LIN {X 0,Y 290.409,Z 885.238,A -85,B 0,C 180,E1 14491.775,E2 14491.775} C_VEL
LIN {X 0,Y 290.448,Z 885.193,A -85,B 0,C 180,E1 14487.632,E2 14487.632} C_VEL
LIN {X 0,Y 290.881,Z 883.624,A -85,B 0,C 180,E1 14483.487,E2 14483.487} C_VEL
LIN {X 0,Y 291.889,Z 880.575,A -85,B 0,C 180,E1 14479.341,E2 14479.341} C_VEL
LIN {X 0,Y 293.714,Z 875.67,A -85,B 0,C 180,E1 14475.007,E2 14475.007} C_VEL
LIN {X 0,Y 296.27,Z 869.554,A -85,B 0,C 180,E1 14471.097,E2 14471.097} C_VEL
LIN {X 0,Y 299.729,Z 861.682,A -85,B 0,C 180,E1 14467.236,E2 14467.236} C_VEL
LIN {X 0,Y 304.292,Z 851.484,A -85,B 0,C 180,E1 14463.349,E2 14463.349} C_VEL
LIN {X 0,Y 309.291,Z 840.18,A -85,B 0,C 180,E1 14459.931,E2 14459.931} C_VEL
LIN {X 0,Y 314.618,Z 827.702,A -85,B 0,C 180,E1 14456.868,E2 14456.868} C_VEL
LIN {X 0,Y 320.27,Z 813.754,A -85,B 0,C 180,E1 14454.065,E2 14454.065} C_VEL
LIN {X 0,Y 325.878,Z 798.802,A -85,B 0,C 180,E1 14451.592,E2 14451.592} C_VEL
LIN {X 0,Y 326.277,Z 797.642,A -85,B 0,C 180,E1 14451.422,E2 14451.422} C_VEL
LIN {X 0,Y 327.524,Z 792.143,A -85,B 0,C 180,E1 14450.493,E2 14450.493} C_VEL
LIN {X 0,Y 328.002,Z 778.328,A -85,B 0,C 180,E1 14447.929,E2 14447.929} C_VEL
LIN {X 0,Y 329.187,Z 772.235,A -85,B 0,C 180,E1 14447.122,E2 14447.122} C_VEL
LIN {X 0,Y 334.318,Z 754.064,A -85,B 0,C 180,E1 14445.351,E2 14445.351} C_VEL
LIN {X 0,Y 338.615,Z 735.624,A -85,B 0,C 180,E1 14443.911,E2 14443.911} C_VEL
LIN {X 0,Y 342.229,Z 716.359,A -85,B 0,C 180,E1 14442.716,E2 14442.716} C_VEL
LIN {X 0,Y 345.103,Z 695.919,A -85,B 0,C 180,E1 14441.743,E2 14441.743} C_VEL
LIN {X 0,Y 346.998,Z 675.756,A -85,B 0,C 180,E1 14441.046,E2 14441.046} C_VEL
LIN {X 0,Y 349.676,Z 625.674,A -85,B 0,C 180,E1 14439.978,E2 14439.978} C_VEL
LIN {X 0,Y 357.062,Z 493.743,A -85,B 0,C 180,E1 14437.345,E2 14437.345} C_VEL
LIN {X 0,Y 348.869,Z 480.651,A -85,B 0,C 180,E1 14434.824,E2 14434.824} C_VEL
LIN {X 0,Y 340.95,Z 468.944,A -85,B 0,C 180,E1 14432.109,E2 14432.109} C_VEL
LIN {X 0,Y 333.261,Z 458.594,A -85,B 0,C 180,E1 14429.13,E2 14429.13} C_VEL
LIN {X 0,Y 329.157,Z 453.339,A -85,B 0,C 180,E1 14427.352,E2 14427.352} C_VEL
LIN {X 0,Y 325.768,Z 449.026,A -85,B 0,C 180,E1 14425.741,E2 14425.741} C_VEL
LIN {X 0,Y 321.751,Z 444.067,A -85,B 0,C 180,E1 14423.633,E2 14423.633} C_VEL
LIN {X 0,Y 317.156,Z 438.642,A -85,B 0,C 180,E1 14420.87,E2 14420.87} C_VEL
LIN {X 0,Y 313.204,Z 434.22,A -85,B 0,C 180,E1 14418.039,E2 14418.039} C_VEL
LIN {X 0,Y 311.897,Z 432.781,A -85,B 0,C 180,E1 14416.961,E2 14416.961} C_VEL
LIN {X 0,Y 306.235,Z 426.851,A -85,B 0,C 180,E1 14410.536,E2 14410.536} C_VEL
LIN {X 0,Y 304.093,Z 425.512,A -85,B 0,C 180,E1 14405.012,E2 14405.012} C_VEL
LIN {X 0,Y 304.604,Z 426.367,A -85,B 0,C 180,E1 14399.248,E2 14399.248} C_VEL
LIN {X 0,Y 308.994,Z 432.434,A -85,B 0,C 180,E1 14392.096,E2 14392.096} C_VEL
LIN {X 0,Y 312.085,Z 436.892,A -85,B 0,C 180,E1 14389.105,E2 14389.105} C_VEL
LIN {X 0,Y 313.416,Z 438.523,A -85,B 0,C 180,E1 14388.033,E2 14388.033} C_VEL
LIN {X 0,Y 317.449,Z 443.877,A -85,B 0,C 180,E1 14385.173,E2 14385.173} C_VEL
LIN {X 0,Y 322.042,Z 450.238,A -85,B 0,C 180,E1 14382.427,E2 14382.427} C_VEL
LIN {X 0,Y 325.886,Z 455.636,A -85,B 0,C 180,E1 14380.416,E2 14380.416} C_VEL
LIN {X 0,Y 329.975,Z 461.384,A -85,B 0,C 180,E1 14378.492,E2 14378.492} C_VEL
LIN {X 0,Y 337.184,Z 472.131,A -85,B 0,C 180,E1 14375.472,E2 14375.472} C_VEL
LIN {X 0,Y 345.291,Z 485.16,A -85,B 0,C 180,E1 14372.493,E2 14372.493} C_VEL
LIN {X 0,Y 353.679,Z 499.744,A -85,B 0,C 180,E1 14369.741,E2 14369.741} C_VEL
LIN {X 0,Y 358.79,Z 509.616,A -85,B 0,C 180,E1 14368.177,E2 14368.177} C_VEL
LIN {X 0,Y 345.156,Z 726.934,A -85,B 0,C 180,E1 14363.563,E2 14363.563} C_VEL
LIN {X 0,Y 342.592,Z 750.271,A -85,B 0,C 180,E1 14362.89,E2 14362.89} C_VEL
LIN {X 0,Y 339.061,Z 771.428,A -85,B 0,C 180,E1 14362.078,E2 14362.078} C_VEL
LIN {X 0,Y 334.52,Z 792.579,A -85,B 0,C 180,E1 14360.992,E2 14360.992} C_VEL
LIN {X 0,Y 329.38,Z 812.962,A -85,B 0,C 180,E1 14359.629,E2 14359.629} C_VEL
LIN {X 0,Y 323.471,Z 833.709,A -85,B 0,C 180,E1 14357.875,E2 14357.875} C_VEL
LIN {X 0,Y 317.514,Z 852.768,A -85,B 0,C 180,E1 14355.883,E2 14355.883} C_VEL
LIN {X 0,Y 311.126,Z 871.664,A -85,B 0,C 180,E1 14353.446,E2 14353.446} C_VEL
LIN {X 0,Y 305.032,Z 889.034,A -85,B 0,C 180,E1 14350.711,E2 14350.711} C_VEL
LIN {X 0,Y 298.988,Z 905.992,A -85,B 0,C 180,E1 14347.487,E2 14347.487} C_VEL
LIN {X 0,Y 293.913,Z 920.626,A -85,B 0,C 180,E1 14344.143,E2 14344.143} C_VEL
LIN {X 0,Y 289.56,Z 933.897,A -85,B 0,C 180,E1 14340.501,E2 14340.501} C_VEL
LIN {X 0,Y 286.009,Z 946,A -85,B 0,C 180,E1 14336.499,E2 14336.499} C_VEL
LIN {X 0,Y 283.419,Z 956.775,A -85,B 0,C 180,E1 14332.176,E2 14332.176} C_VEL
LIN {X 0,Y 281.949,Z 965.312,A -85,B 0,C 180,E1 14327.969,E2 14327.969} C_VEL
LIN {X 0,Y 281.351,Z 971.642,A -85,B 0,C 180,E1 14323.984,E2 14323.984} C_VEL
LIN {X 0,Y 281.318,Z 976.689,A -85,B 0,C 180,E1 14319.822,E2 14319.822} C_VEL
LIN {X 0,Y 281.574,Z 979.725,A -85,B 0,C 180,E1 14316.115,E2 14316.115} C_VEL
LIN {X 0,Y 281.797,Z 981.427,A -85,B 0,C 180,E1 14312.441,E2 14312.441} C_VEL
LIN {X 0,Y 281.86,Z 981.636,A -85,B 0,C 180,E1 14308.985,E2 14308.985} C_VEL
LIN {X 0,Y 281.703,Z 980.723,A -85,B 0,C 180,E1 14305.727,E2 14305.727} C_VEL
LIN {X 0,Y 281.41,Z 978.219,A -85,B 0,C 180,E1 14301.831,E2 14301.831} C_VEL
LIN {X 0,Y 281.285,Z 974.359,A -85,B 0,C 180,E1 14298.104,E2 14298.104} C_VEL
LIN {X 0,Y 281.594,Z 968.491,A -85,B 0,C 180,E1 14293.924,E2 14293.924} C_VEL
LIN {X 0,Y 282.637,Z 960.839,A -85,B 0,C 180,E1 14289.718,E2 14289.718} C_VEL
LIN {X 0,Y 284.644,Z 951.268,A -85,B 0,C 180,E1 14285.516,E2 14285.516} C_VEL
LIN {X 0,Y 287.76,Z 939.735,A -85,B 0,C 180,E1 14281.351,E2 14281.351} C_VEL
LIN {X 0,Y 291.612,Z 927.517,A -85,B 0,C 180,E1 14277.669,E2 14277.669} C_VEL
LIN {X 0,Y 296.576,Z 912.818,A -85,B 0,C 180,E1 14274.009,E2 14274.009} C_VEL
LIN {X 0,Y 302.138,Z 897.046,A -85,B 0,C 180,E1 14270.747,E2 14270.747} C_VEL
LIN {X 0,Y 308.386,Z 879.4,A -85,B 0,C 180,E1 14267.726,E2 14267.726} C_VEL
LIN {X 0,Y 314.378,Z 862.063,A -85,B 0,C 180,E1 14265.267,E2 14265.267} C_VEL
LIN {X 0,Y 320.426,Z 843.454,A -85,B 0,C 180,E1 14263.106,E2 14263.106} C_VEL
LIN {X 0,Y 326.091,Z 824.547,A -85,B 0,C 180,E1 14261.312,E2 14261.312} C_VEL
LIN {X 0,Y 331.598,Z 804.213,A -85,B 0,C 180,E1 14259.753,E2 14259.753} C_VEL
LIN {X 0,Y 336.584,Z 783.168,A -85,B 0,C 180,E1 14258.495,E2 14258.495} C_VEL
LIN {X 0,Y 340.77,Z 761.554,A -85,B 0,C 180,E1 14257.53,E2 14257.53} C_VEL
LIN {X 0,Y 343.932,Z 738.988,A -85,B 0,C 180,E1 14256.768,E2 14256.768} C_VEL
LIN {X 0,Y 346.033,Z 712.945,A -85,B 0,C 180,E1 14256.132,E2 14256.132} C_VEL
LIN {X 0,Y 358.699,Z 509.365,A -85,B 0,C 180,E1 14251.827,E2 14251.827} C_VEL
LIN {X 0,Y 349.918,Z 493.137,A -85,B 0,C 180,E1 14249.109,E2 14249.109} C_VEL
LIN {X 0,Y 341.866,Z 479.602,A -85,B 0,C 180,E1 14246.348,E2 14246.348} C_VEL
LIN {X 0,Y 335.259,Z 469.393,A -85,B 0,C 180,E1 14243.835,E2 14243.835} C_VEL
LIN {X 0,Y 327.618,Z 457.902,A -85,B 0,C 180,E1 14240.499,E2 14240.499} C_VEL
LIN {X 0,Y 320.59,Z 448.147,A -85,B 0,C 180,E1 14236.86,E2 14236.86} C_VEL
LIN {X 0,Y 316.137,Z 442.173,A -85,B 0,C 180,E1 14234.095,E2 14234.095} C_VEL
LIN {X 0,Y 312.318,Z 437.185,A -85,B 0,C 180,E1 14231.261,E2 14231.261} C_VEL
LIN {X 0,Y 309.021,Z 432.656,A -85,B 0,C 180,E1 14228.184,E2 14228.184} C_VEL
LIN {X 0,Y 308.029,Z 431.411,A -85,B 0,C 180,E1 14227.085,E2 14227.085} C_VEL
LIN {X 0,Y 304.423,Z 426.254,A -85,B 0,C 180,E1 14220.941,E2 14220.941} C_VEL
LIN {X 0,Y 303.838,Z 425.332,A -85,B 0,C 180,E1 14214.902,E2 14214.902} C_VEL
LIN {X 0,Y 305.725,Z 426.487,A -85,B 0,C 180,E1 14209.828,E2 14209.828} C_VEL
LIN {X 0,Y 307.208,Z 427.964,A -85,B 0,C 180,E1 14207.595,E2 14207.595} C_VEL
LIN {X 0,Y 312.808,Z 433.677,A -85,B 0,C 180,E1 14202.034,E2 14202.034} C_VEL
LIN {X 0,Y 316.844,Z 438.399,A -85,B 0,C 180,E1 14199.109,E2 14199.109} C_VEL
LIN {X 0,Y 318.218,Z 439.909,A -85,B 0,C 180,E1 14198.237,E2 14198.237} C_VEL
LIN {X 0,Y 322.234,Z 444.497,A -85,B 0,C 180,E1 14195.918,E2 14195.918} C_VEL
LIN {X 0,Y 327.796,Z 451.607,A -85,B 0,C 180,E1 14193.115,E2 14193.115} C_VEL
LIN {X 0,Y 332.097,Z 457.141,A -85,B 0,C 180,E1 14191.202,E2 14191.202} C_VEL
LIN {X 0,Y 338.239,Z 465.249,A -85,B 0,C 180,E1 14188.748,E2 14188.748} C_VEL
LIN {X 0,Y 346.862,Z 477.634,A -85,B 0,C 180,E1 14185.698,E2 14185.698} C_VEL
LIN {X 0,Y 355.474,Z 491.21,A -85,B 0,C 180,E1 14182.992,E2 14182.992} C_VEL
LIN {X 0,Y 357.054,Z 494.161,A -85,B 0,C 180,E1 14182.515,E2 14182.515} C_VEL
LIN {X 0,Y 347.059,Z 672.789,A -85,B 0,C 180,E1 14178.93,E2 14178.93} C_VEL
LIN {X 0,Y 345.224,Z 693.984,A -85,B 0,C 180,E1 14178.232,E2 14178.232} C_VEL
LIN {X 0,Y 342.488,Z 714.257,A -85,B 0,C 180,E1 14177.297,E2 14177.297} C_VEL
LIN {X 0,Y 339.005,Z 733.494,A -85,B 0,C 180,E1 14176.136,E2 14176.136} C_VEL
LIN {X 0,Y 334.567,Z 752.673,A -85,B 0,C 180,E1 14174.661,E2 14174.661} C_VEL
LIN {X 0,Y 329.766,Z 769.978,A -85,B 0,C 180,E1 14173.01,E2 14173.01} C_VEL
LIN {X 0,Y 324.127,Z 787.653,A -85,B 0,C 180,E1 14170.941,E2 14170.941} C_VEL
LIN {X 0,Y 318.438,Z 803.532,A -85,B 0,C 180,E1 14168.665,E2 14168.665} C_VEL
LIN {X 0,Y 312.517,Z 818.483,A -85,B 0,C 180,E1 14166.059,E2 14166.059} C_VEL
LIN {X 0,Y 306.776,Z 831.838,A -85,B 0,C 180,E1 14163.195,E2 14163.195} C_VEL
LIN {X 0,Y 301.346,Z 843.808,A -85,B 0,C 180,E1 14160.063,E2 14160.063} C_VEL
LIN {X 0,Y 296.149,Z 854.942,A -85,B 0,C 180,E1 14156.462,E2 14156.462} C_VEL
LIN {X 0,Y 291.874,Z 864.064,A -85,B 0,C 180,E1 14152.771,E2 14152.771} C_VEL
LIN {X 0,Y 288.37,Z 871.774,A -85,B 0,C 180,E1 14148.809,E2 14148.809} C_VEL
LIN {X 0,Y 285.67,Z 877.943,A -85,B 0,C 180,E1 14144.594,E2 14144.594} C_VEL
LIN {X 0,Y 283.939,Z 882.349,A -85,B 0,C 180,E1 14140.344,E2 14140.344} C_VEL
LIN {X 0,Y 282.94,Z 885.19,A -85,B 0,C 180,E1 14136.084,E2 14136.084} C_VEL
LIN {X 0,Y 282.523,Z 886.567,A -85,B 0,C 180,E1 14131.824,E2 14131.824} C_VEL
LIN {X 0,Y 282.563,Z 886.521,A -85,B 0,C 180,E1 14127.566,E2 14127.566} C_VEL
LIN {X 0,Y 283.03,Z 884.955,A -85,B 0,C 180,E1 14123.305,E2 14123.305} C_VEL
LIN {X 0,Y 284.108,Z 881.909,A -85,B 0,C 180,E1 14119.045,E2 14119.045} C_VEL
LIN {X 0,Y 286.058,Z 877.01,A -85,B 0,C 180,E1 14114.596,E2 14114.596} C_VEL
LIN {X 0,Y 288.767,Z 870.9,A -85,B 0,C 180,E1 14110.587,E2 14110.587} C_VEL
LIN {X 0,Y 292.425,Z 863.031,A -85,B 0,C 180,E1 14106.634,E2 14106.634} C_VEL
LIN {X 0,Y 297.085,Z 853.112,A -85,B 0,C 180,E1 14102.762,E2 14102.762} C_VEL
LIN {X 0,Y 302.17,Z 842.154,A -85,B 0,C 180,E1 14099.353,E2 14099.353} C_VEL
LIN {X 0,Y 307.678,Z 829.872,A -85,B 0,C 180,E1 14096.244,E2 14096.244} C_VEL
LIN {X 0,Y 313.527,Z 816.113,A -85,B 0,C 180,E1 14093.394,E2 14093.394} C_VEL
LIN {X 0,Y 319.335,Z 801.393,A -85,B 0,C 180,E1 14090.887,E2 14090.887} C_VEL
LIN {X 0,Y 325.122,Z 785.032,A -85,B 0,C 180,E1 14088.613,E2 14088.613} C_VEL
LIN {X 0,Y 329.187,Z 772.235,A -85,B 0,C 180,E1 14087.122,E2 14087.122} C_VEL
LIN {X 0,Y 330.457,Z 765.992,A -85,B 0,C 180,E1 14086.346,E2 14086.346} C_VEL
LIN {X 0,Y 330.75,Z 750.626,A -85,B 0,C 180,E1 14084.094,E2 14084.094} C_VEL
LIN {X 0,Y 331.712,Z 743.976,A -85,B 0,C 180,E1 14083.429,E2 14083.429} C_VEL
LIN {X 0,Y 335.725,Z 725.177,A -85,B 0,C 180,E1 14082.14,E2 14082.14} C_VEL
LIN {X 0,Y 338.968,Z 705.436,A -85,B 0,C 180,E1 14081.084,E2 14081.084} C_VEL
LIN {X 0,Y 341.414,Z 684.411,A -85,B 0,C 180,E1 14080.253,E2 14080.253} C_VEL
LIN {X 0,Y 342.879,Z 662.381,A -85,B 0,C 180,E1 14079.658,E2 14079.658} C_VEL
LIN {X 0,Y 352.377,Z 497.735,A -85,B 0,C 180,E1 14076.345,E2 14076.345} C_VEL
LIN {X 0,Y 343.887,Z 484.113,A -85,B 0,C 180,E1 14073.584,E2 14073.584} C_VEL
LIN {X 0,Y 335.378,Z 471.633,A -85,B 0,C 180,E1 14070.453,E2 14070.453} C_VEL
LIN {X 0,Y 327.784,Z 461.467,A -85,B 0,C 180,E1 14067.23,E2 14067.23} C_VEL
LIN {X 0,Y 323.657,Z 456.225,A -85,B 0,C 180,E1 14065.234,E2 14065.234} C_VEL
LIN {X 0,Y 319.892,Z 451.487,A -85,B 0,C 180,E1 14063.193,E2 14063.193} C_VEL
LIN {X 0,Y 315.547,Z 446.233,A -85,B 0,C 180,E1 14060.496,E2 14060.496} C_VEL
LIN {X 0,Y 311.599,Z 441.616,A -85,B 0,C 180,E1 14057.556,E2 14057.556} C_VEL
LIN {X 0,Y 309.905,Z 440.067,A -85,B 0,C 180,E1 14056.109,E2 14056.109} C_VEL
LIN {X 0,Y 305.169,Z 434.743,A -85,B 0,C 180,E1 14050.382,E2 14050.382} C_VEL
LIN {X 0,Y 303.105,Z 433.451,A -85,B 0,C 180,E1 14044.921,E2 14044.921} C_VEL
LIN {X 0,Y 303.611,Z 434.332,A -85,B 0,C 180,E1 14039.246,E2 14039.246} C_VEL
LIN {X 0,Y 307.728,Z 440.294,A -85,B 0,C 180,E1 14032.345,E2 14032.345} C_VEL
LIN {X 0,Y 310.977,Z 444.898,A -85,B 0,C 180,E1 14029.159,E2 14029.159} C_VEL
LIN {X 0,Y 315.697,Z 451.327,A -85,B 0,C 180,E1 14025.605,E2 14025.605} C_VEL
LIN {X 0,Y 320.403,Z 458.009,A -85,B 0,C 180,E1 14022.709,E2 14022.709} C_VEL
LIN {X 0,Y 325.963,Z 465.865,A -85,B 0,C 180,E1 14019.814,E2 14019.814} C_VEL
LIN {X 0,Y 333.477,Z 477.362,A -85,B 0,C 180,E1 14016.452,E2 14016.452} C_VEL
LIN {X 0,Y 339.968,Z 487.805,A -85,B 0,C 180,E1 14013.917,E2 14013.917} C_VEL
LIN {X 0,Y 347.35,Z 500.6,A -85,B 0,C 180,E1 14011.315,E2 14011.315} C_VEL
LIN {X 0,Y 353.993,Z 513.293,A -85,B 0,C 180,E1 14009.161,E2 14009.161} C_VEL
LIN {X 0,Y 340.097,Z 726.961,A -85,B 0,C 180,E1 14004.602,E2 14004.602} C_VEL
LIN {X 0,Y 337.422,Z 750.06,A -85,B 0,C 180,E1 14003.925,E2 14003.925} C_VEL
LIN {X 0,Y 333.61,Z 771.835,A -85,B 0,C 180,E1 14003.073,E2 14003.073} C_VEL
LIN {X 0,Y 328.817,Z 793.371,A -85,B 0,C 180,E1 14001.952,E2 14001.952} C_VEL
LIN {X 0,Y 323.524,Z 813.342,A -85,B 0,C 180,E1 14000.585,E2 14000.585} C_VEL
LIN {X 0,Y 317.443,Z 833.743,A -85,B 0,C 180,E1 13998.826,E2 13998.826} C_VEL
LIN {X 0,Y 311.264,Z 852.623,A -85,B 0,C 180,E1 13996.813,E2 13996.813} C_VEL
LIN {X 0,Y 304.638,Z 871.415,A -85,B 0,C 180,E1 13994.349,E2 13994.349} C_VEL
LIN {X 0,Y 298.296,Z 888.614,A -85,B 0,C 180,E1 13991.577,E2 13991.577} C_VEL
LIN {X 0,Y 292.146,Z 904.974,A -85,B 0,C 180,E1 13988.396,E2 13988.396} C_VEL
LIN {X 0,Y 286.666,Z 919.933,A -85,B 0,C 180,E1 13984.888,E2 13984.888} C_VEL
LIN {X 0,Y 282.089,Z 933.143,A -85,B 0,C 180,E1 13981.162,E2 13981.162} C_VEL
LIN {X 0,Y 278.396,Z 944.932,A -85,B 0,C 180,E1 13977.135,E2 13977.135} C_VEL
LIN {X 0,Y 275.596,Z 955.82,A -85,B 0,C 180,E1 13972.615,E2 13972.615} C_VEL
LIN {X 0,Y 274.039,Z 964.27,A -85,B 0,C 180,E1 13968.286,E2 13968.286} C_VEL
LIN {X 0,Y 273.401,Z 970.56,A -85,B 0,C 180,E1 13964.183,E2 13964.183} C_VEL
LIN {X 0,Y 273.386,Z 975.525,A -85,B 0,C 180,E1 13959.898,E2 13959.898} C_VEL
LIN {X 0,Y 273.641,Z 978.381,A -85,B 0,C 180,E1 13956.293,E2 13956.293} C_VEL
LIN {X 0,Y 273.901,Z 980.097,A -85,B 0,C 180,E1 13952.511,E2 13952.511} C_VEL
LIN {X 0,Y 273.971,Z 980.307,A -85,B 0,C 180,E1 13948.955,E2 13948.955} C_VEL
LIN {X 0,Y 273.789,Z 979.36,A -85,B 0,C 180,E1 13945.537,E2 13945.537} C_VEL
LIN {X 0,Y 273.466,Z 976.864,A -85,B 0,C 180,E1 13941.592,E2 13941.592} C_VEL
LIN {X 0,Y 273.34,Z 972.987,A -85,B 0,C 180,E1 13937.753,E2 13937.753} C_VEL
LIN {X 0,Y 273.736,Z 966.743,A -85,B 0,C 180,E1 13933.231,E2 13933.231} C_VEL
LIN {X 0,Y 274.932,Z 959.016,A -85,B 0,C 180,E1 13928.901,E2 13928.901} C_VEL
LIN {X 0,Y 277.167,Z 949.314,A -85,B 0,C 180,E1 13924.582,E2 13924.582} C_VEL
LIN {X 0,Y 280.579,Z 937.642,A -85,B 0,C 180,E1 13920.312,E2 13920.312} C_VEL
LIN {X 0,Y 285.012,Z 924.508,A -85,B 0,C 180,E1 13916.343,E2 13916.343} C_VEL
LIN {X 0,Y 290.333,Z 909.936,A -85,B 0,C 180,E1 13912.696,E2 13912.696} C_VEL
LIN {X 0,Y 296.32,Z 893.776,A -85,B 0,C 180,E1 13909.371,E2 13909.371} C_VEL
LIN {X 0,Y 302.646,Z 876.69,A -85,B 0,C 180,E1 13906.469,E2 13906.469} C_VEL
LIN {X 0,Y 309.294,Z 858.127,A -85,B 0,C 180,E1 13903.878,E2 13903.878} C_VEL
LIN {X 0,Y 315.572,Z 839.508,A -85,B 0,C 180,E1 13901.749,E2 13901.749} C_VEL
LIN {X 0,Y 321.813,Z 819.166,A -85,B 0,C 180,E1 13899.885,E2 13899.885} C_VEL
LIN {X 0,Y 327.168,Z 799.467,A -85,B 0,C 180,E1 13898.45,E2 13898.45} C_VEL
LIN {X 0,Y 332.218,Z 778.146,A -85,B 0,C 180,E1 13897.24,E2 13897.24} C_VEL
LIN {X 0,Y 336.389,Z 756.516,A -85,B 0,C 180,E1 13896.311,E2 13896.311} C_VEL
LIN {X 0,Y 339.397,Z 733.736,A -85,B 0,C 180,E1 13895.583,E2 13895.583} C_VEL
LIN {X 0,Y 342.016,Z 697.121,A -85,B 0,C 180,E1 13894.748,E2 13894.748} C_VEL
LIN {X 0,Y 353.853,Z 513.011,A -85,B 0,C 180,E1 13890.83,E2 13890.83} C_VEL
LIN {X 0,Y 346.128,Z 498.547,A -85,B 0,C 180,E1 13888.324,E2 13888.324} C_VEL
LIN {X 0,Y 338.507,Z 485.449,A -85,B 0,C 180,E1 13885.593,E2 13885.593} C_VEL
LIN {X 0,Y 330.804,Z 473.239,A -85,B 0,C 180,E1 13882.479,E2 13882.479} C_VEL
LIN {X 0,Y 324.449,Z 463.863,A -85,B 0,C 180,E1 13879.533,E2 13879.533} C_VEL
LIN {X 0,Y 319.858,Z 457.309,A -85,B 0,C 180,E1 13877.087,E2 13877.087} C_VEL
LIN {X 0,Y 314.488,Z 449.707,A -85,B 0,C 180,E1 13873.701,E2 13873.701} C_VEL
LIN {X 0,Y 310.772,Z 444.756,A -85,B 0,C 180,E1 13870.848,E2 13870.848} C_VEL
LIN {X 0,Y 307.604,Z 440.178,A -85,B 0,C 180,E1 13867.752,E2 13867.752} C_VEL
LIN {X 0,Y 303.444,Z 434.221,A -85,B 0,C 180,E1 13860.944,E2 13860.944} C_VEL
LIN {X 0,Y 302.837,Z 433.273,A -85,B 0,C 180,E1 13855.075,E2 13855.075} C_VEL
LIN {X 0,Y 304.552,Z 434.314,A -85,B 0,C 180,E1 13850.17,E2 13850.17} C_VEL
LIN {X 0,Y 305.983,Z 435.681,A -85,B 0,C 180,E1 13847.928,E2 13847.928} C_VEL
LIN {X 0,Y 311.415,Z 441.399,A -85,B 0,C 180,E1 13842.337,E2 13842.337} C_VEL
LIN {X 0,Y 315.506,Z 446.218,A -85,B 0,C 180,E1 13839.307,E2 13839.307} C_VEL
LIN {X 0,Y 317.527,Z 448.87,A -85,B 0,C 180,E1 13837.993,E2 13837.993} C_VEL
LIN {X 0,Y 321.204,Z 453.087,A -85,B 0,C 180,E1 13835.885,E2 13835.885} C_VEL
LIN {X 0,Y 325.897,Z 459.13,A -85,B 0,C 180,E1 13833.487,E2 13833.487} C_VEL
LIN {X 0,Y 330.217,Z 464.811,A -85,B 0,C 180,E1 13831.517,E2 13831.517} C_VEL
LIN {X 0,Y 336.271,Z 473.07,A -85,B 0,C 180,E1 13829.043,E2 13829.043} C_VEL
LIN {X 0,Y 343.904,Z 484.236,A -85,B 0,C 180,E1 13826.268,E2 13826.268} C_VEL
LIN {X 0,Y 352.379,Z 497.846,A -85,B 0,C 180,E1 13823.52,E2 13823.52} C_VEL
LIN {X 0,Y 342.143,Z 673.459,A -85,B 0,C 180,E1 13819.973,E2 13819.973} C_VEL
LIN {X 0,Y 340.24,Z 694.769,A -85,B 0,C 180,E1 13819.27,E2 13819.27} C_VEL
LIN {X 0,Y 337.483,Z 714.678,A -85,B 0,C 180,E1 13818.353,E2 13818.353} C_VEL
LIN {X 0,Y 333.79,Z 734.452,A -85,B 0,C 180,E1 13817.158,E2 13817.158} C_VEL
LIN {X 0,Y 329.272,Z 753.343,A -85,B 0,C 180,E1 13815.7,E2 13815.7} C_VEL
LIN {X 0,Y 324.306,Z 770.719,A -85,B 0,C 180,E1 13814.039,E2 13814.039} C_VEL
LIN {X 0,Y 318.477,Z 788.412,A -85,B 0,C 180,E1 13811.962,E2 13811.962} C_VEL
LIN {X 0,Y 312.75,Z 803.9,A -85,B 0,C 180,E1 13809.741,E2 13809.741} C_VEL
LIN {X 0,Y 306.564,Z 818.95,A -85,B 0,C 180,E1 13807.107,E2 13807.107} C_VEL
LIN {X 0,Y 300.537,Z 832.432,A -85,B 0,C 180,E1 13804.207,E2 13804.207} C_VEL
LIN {X 0,Y 294.83,Z 844.524,A -85,B 0,C 180,E1 13801.025,E2 13801.025} C_VEL
LIN {X 0,Y 289.602,Z 855.245,A -85,B 0,C 180,E1 13797.554,E2 13797.554} C_VEL
LIN {X 0,Y 285.012,Z 864.578,A -85,B 0,C 180,E1 13793.79,E2 13793.79} C_VEL
LIN {X 0,Y 281.027,Z 872.781,A -85,B 0,C 180,E1 13789.536,E2 13789.536} C_VEL
LIN {X 0,Y 278.114,Z 879.014,A -85,B 0,C 180,E1 13785.213,E2 13785.213} C_VEL
LIN {X 0,Y 276.219,Z 883.504,A -85,B 0,C 180,E1 13780.848,E2 13780.848} C_VEL
LIN {X 0,Y 275.084,Z 886.521,A -85,B 0,C 180,E1 13776.259,E2 13776.259} C_VEL
LIN {X 0,Y 274.637,Z 887.895,A -85,B 0,C 180,E1 13771.877,E2 13771.877} C_VEL
LIN {X 0,Y 274.679,Z 887.849,A -85,B 0,C 180,E1 13767.496,E2 13767.496} C_VEL
LIN {X 0,Y 275.181,Z 886.285,A -85,B 0,C 180,E1 13763.113,E2 13763.113} C_VEL
LIN {X 0,Y 276.36,Z 883.18,A -85,B 0,C 180,E1 13758.659,E2 13758.659} C_VEL
LIN {X 0,Y 278.417,Z 878.349,A -85,B 0,C 180,E1 13754.162,E2 13754.162} C_VEL
LIN {X 0,Y 281.287,Z 872.246,A -85,B 0,C 180,E1 13750.049,E2 13750.049} C_VEL
LIN {X 0,Y 285.154,Z 864.379,A -85,B 0,C 180,E1 13746.002,E2 13746.002} C_VEL
LIN {X 0,Y 290.053,Z 854.464,A -85,B 0,C 180,E1 13742.045,E2 13742.045} C_VEL
LIN {X 0,Y 295.361,Z 843.557,A -85,B 0,C 180,E1 13738.582,E2 13738.582} C_VEL
LIN {X 0,Y 301.132,Z 831.251,A -85,B 0,C 180,E1 13735.408,E2 13735.408} C_VEL
LIN {X 0,Y 307.226,Z 817.514,A -85,B 0,C 180,E1 13732.516,E2 13732.516} C_VEL
LIN {X 0,Y 313.14,Z 803.132,A -85,B 0,C 180,E1 13730.025,E2 13730.025} C_VEL
LIN {X 0,Y 319.027,Z 787.123,A -85,B 0,C 180,E1 13727.763,E2 13727.763} C_VEL
LIN {X 0,Y 324.643,Z 769.911,A -85,B 0,C 180,E1 13725.771,E2 13725.771} C_VEL
LIN {X 0,Y 329.998,Z 750.81,A -85,B 0,C 180,E1 13723.984,E2 13723.984} C_VEL
LIN {X 0,Y 331.712,Z 743.976,A -85,B 0,C 180,E1 13723.429,E2 13723.429} C_VEL
LIN {X 0,Y 332.656,Z 737.184,A -85,B 0,C 180,E1 13722.796,E2 13722.796} C_VEL
LIN {X 0,Y 332.414,Z 720.417,A -85,B 0,C 180,E1 13720.883,E2 13720.883} C_VEL
LIN {X 0,Y 333.007,Z 713.325,A -85,B 0,C 180,E1 13720.358,E2 13720.358} C_VEL
LIN {X 0,Y 335.84,Z 692.533,A -85,B 0,C 180,E1 13719.437,E2 13719.437} C_VEL
LIN {X 0,Y 337.59,Z 671.891,A -85,B 0,C 180,E1 13718.792,E2 13718.792} C_VEL
LIN {X 0,Y 347.809,Z 501.843,A -85,B 0,C 180,E1 13715.324,E2 13715.324} C_VEL
LIN {X 0,Y 339.689,Z 488.749,A -85,B 0,C 180,E1 13712.542,E2 13712.542} C_VEL
LIN {X 0,Y 332.452,Z 478.055,A -85,B 0,C 180,E1 13709.752,E2 13709.752} C_VEL
LIN {X 0,Y 325.609,Z 468.642,A -85,B 0,C 180,E1 13706.735,E2 13706.735} C_VEL
LIN {X 0,Y 321.573,Z 463.42,A -85,B 0,C 180,E1 13704.721,E2 13704.721} C_VEL
LIN {X 0,Y 318.053,Z 458.904,A -85,B 0,C 180,E1 13702.748,E2 13702.748} C_VEL
LIN {X 0,Y 313.952,Z 453.821,A -85,B 0,C 180,E1 13700.118,E2 13700.118} C_VEL
LIN {X 0,Y 310.015,Z 449.017,A -85,B 0,C 180,E1 13697.068,E2 13697.068} C_VEL
LIN {X 0,Y 304.101,Z 442.634,A -85,B 0,C 180,E1 13690.227,E2 13690.227} C_VEL
LIN {X 0,Y 302.133,Z 441.392,A -85,B 0,C 180,E1 13684.936,E2 13684.936} C_VEL
LIN {X 0,Y 302.575,Z 442.213,A -85,B 0,C 180,E1 13679.432,E2 13679.432} C_VEL
LIN {X 0,Y 306.397,Z 447.98,A -85,B 0,C 180,E1 13672.689,E2 13672.689} C_VEL
LIN {X 0,Y 309.653,Z 452.685,A -85,B 0,C 180,E1 13669.395,E2 13669.395} C_VEL
LIN {X 0,Y 314.024,Z 458.88,A -85,B 0,C 180,E1 13665.997,E2 13665.997} C_VEL
LIN {X 0,Y 318.476,Z 465.346,A -85,B 0,C 180,E1 13663.165,E2 13663.165} C_VEL
LIN {X 0,Y 323.903,Z 473.259,A -85,B 0,C 180,E1 13660.244,E2 13660.244} C_VEL
LIN {X 0,Y 331.467,Z 485.039,A -85,B 0,C 180,E1 13656.772,E2 13656.772} C_VEL
LIN {X 0,Y 339.288,Z 498.214,A -85,B 0,C 180,E1 13653.672,E2 13653.672} C_VEL
LIN {X 0,Y 346.92,Z 512.19,A -85,B 0,C 180,E1 13650.97,E2 13650.97} C_VEL
LIN {X 0,Y 349.299,Z 517.092,A -85,B 0,C 180,E1 13650.171,E2 13650.171} C_VEL
LIN {X 0,Y 335.185,Z 726.611,A -85,B 0,C 180,E1 13645.682,E2 13645.682} C_VEL
LIN {X 0,Y 332.443,Z 749.345,A -85,B 0,C 180,E1 13645.008,E2 13645.008} C_VEL
LIN {X 0,Y 328.545,Z 770.944,A -85,B 0,C 180,E1 13644.162,E2 13644.162} C_VEL
LIN {X 0,Y 323.816,Z 791.545,A -85,B 0,C 180,E1 13643.097,E2 13643.097} C_VEL
LIN {X 0,Y 318.342,Z 811.649,A -85,B 0,C 180,E1 13641.734,E2 13641.734} C_VEL
LIN {X 0,Y 312.043,Z 832.138,A -85,B 0,C 180,E1 13639.973,E2 13639.973} C_VEL
LIN {X 0,Y 305.623,Z 851.078,A -85,B 0,C 180,E1 13637.951,E2 13637.951} C_VEL
LIN {X 0,Y 298.864,Z 869.411,A -85,B 0,C 180,E1 13635.541,E2 13635.541} C_VEL
LIN {X 0,Y 292.255,Z 886.568,A -85,B 0,C 180,E1 13632.769,E2 13632.769} C_VEL
LIN {X 0,Y 285.763,Z 903.029,A -85,B 0,C 180,E1 13629.55,E2 13629.55} C_VEL
LIN {X 0,Y 280.073,Z 917.7,A -85,B 0,C 180,E1 13626.086,E2 13626.086} C_VEL
LIN {X 0,Y 274.87,Z 931.749,A -85,B 0,C 180,E1 13622.055,E2 13622.055} C_VEL
LIN {X 0,Y 270.927,Z 943.493,A -85,B 0,C 180,E1 13617.947,E2 13617.947} C_VEL
LIN {X 0,Y 267.897,Z 954.4,A -85,B 0,C 180,E1 13613.303,E2 13613.303} C_VEL
LIN {X 0,Y 266.187,Z 962.917,A -85,B 0,C 180,E1 13608.816,E2 13608.816} C_VEL
LIN {X 0,Y 265.464,Z 969.278,A -85,B 0,C 180,E1 13604.541,E2 13604.541} C_VEL
LIN {X 0,Y 265.443,Z 974.165,A -85,B 0,C 180,E1 13600.197,E2 13600.197} C_VEL
LIN {X 0,Y 265.706,Z 977.036,A -85,B 0,C 180,E1 13596.482,E2 13596.482} C_VEL
LIN {X 0,Y 266.005,Z 978.766,A -85,B 0,C 180,E1 13592.586,E2 13592.586} C_VEL
LIN {X 0,Y 266.08,Z 978.979,A -85,B 0,C 180,E1 13588.924,E2 13588.924} C_VEL
LIN {X 0,Y 265.885,Z 978.051,A -85,B 0,C 180,E1 13585.472,E2 13585.472} C_VEL
LIN {X 0,Y 265.519,Z 975.509,A -85,B 0,C 180,E1 13581.338,E2 13581.338} C_VEL
LIN {X 0,Y 265.399,Z 971.584,A -85,B 0,C 180,E1 13577.354,E2 13577.354} C_VEL
LIN {X 0,Y 265.846,Z 965.345,A -85,B 0,C 180,E1 13572.718,E2 13572.718} C_VEL
LIN {X 0,Y 267.173,Z 957.603,A -85,B 0,C 180,E1 13568.257,E2 13568.257} C_VEL
LIN {X 0,Y 269.604,Z 947.881,A -85,B 0,C 180,E1 13563.815,E2 13563.815} C_VEL
LIN {X 0,Y 273.278,Z 936.192,A -85,B 0,C 180,E1 13559.436,E2 13559.436} C_VEL
LIN {X 0,Y 278.004,Z 923.038,A -85,B 0,C 180,E1 13555.376,E2 13555.376} C_VEL
LIN {X 0,Y 283.645,Z 908.454,A -85,B 0,C 180,E1 13551.66,E2 13551.66} C_VEL
LIN {X 0,Y 289.98,Z 892.283,A -85,B 0,C 180,E1 13548.288,E2 13548.288} C_VEL
LIN {X 0,Y 296.382,Z 875.759,A -85,B 0,C 180,E1 13545.443,E2 13545.443} C_VEL
LIN {X 0,Y 303.058,Z 857.974,A -85,B 0,C 180,E1 13542.917,E2 13542.917} C_VEL
LIN {X 0,Y 309.853,Z 838.659,A -85,B 0,C 180,E1 13540.679,E2 13540.679} C_VEL
LIN {X 0,Y 315.995,Z 819.377,A -85,B 0,C 180,E1 13538.895,E2 13538.895} C_VEL
LIN {X 0,Y 321.641,Z 799.53,A -85,B 0,C 180,E1 13537.424,E2 13537.424} C_VEL
LIN {X 0,Y 326.664,Z 779.353,A -85,B 0,C 180,E1 13536.251,E2 13536.251} C_VEL
LIN {X 0,Y 331.065,Z 757.494,A -85,B 0,C 180,E1 13535.295,E2 13535.295} C_VEL
LIN {X 0,Y 334.185,Z 735.532,A -85,B 0,C 180,E1 13534.57,E2 13534.57} C_VEL
LIN {X 0,Y 336.583,Z 705.923,A -85,B 0,C 180,E1 13533.862,E2 13533.862} C_VEL
LIN {X 0,Y 349.187,Z 516.696,A -85,B 0,C 180,E1 13529.824,E2 13529.824} C_VEL
LIN {X 0,Y 340.616,Z 500.647,A -85,B 0,C 180,E1 13526.875,E2 13526.875} C_VEL
LIN {X 0,Y 332.668,Z 487.109,A -85,B 0,C 180,E1 13523.797,E2 13523.797} C_VEL
LIN {X 0,Y 325.553,Z 475.839,A -85,B 0,C 180,E1 13520.635,E2 13520.635} C_VEL
LIN {X 0,Y 319.766,Z 467.155,A -85,B 0,C 180,E1 13517.656,E2 13517.656} C_VEL
LIN {X 0,Y 315.827,Z 461.668,A -85,B 0,C 180,E1 13515.328,E2 13515.328} C_VEL
LIN {X 0,Y 312.737,Z 457.105,A -85,B 0,C 180,E1 13513.214,E2 13513.214} C_VEL
LIN {X 0,Y 309.36,Z 452.436,A -85,B 0,C 180,E1 13510.521,E2 13510.521} C_VEL
LIN {X 0,Y 306.216,Z 447.702,A -85,B 0,C 180,E1 13507.316,E2 13507.316} C_VEL
LIN {X 0,Y 302.404,Z 442.103,A -85,B 0,C 180,E1 13500.757,E2 13500.757} C_VEL
LIN {X 0,Y 301.896,Z 441.214,A -85,B 0,C 180,E1 13494.869,E2 13494.869} C_VEL
LIN {X 0,Y 303.921,Z 442.483,A -85,B 0,C 180,E1 13489.575,E2 13489.575} C_VEL
LIN {X 0,Y 306.159,Z 445.27,A -85,B 0,C 180,E1 13486.4,E2 13486.4} C_VEL
LIN {X 0,Y 310.131,Z 449.278,A -85,B 0,C 180,E1 13482.552,E2 13482.552} C_VEL
LIN {X 0,Y 314.171,Z 454.037,A -85,B 0,C 180,E1 13479.507,E2 13479.507} C_VEL
LIN {X 0,Y 319.559,Z 460.816,A -85,B 0,C 180,E1 13476.195,E2 13476.195} C_VEL
LIN {X 0,Y 323.984,Z 466.612,A -85,B 0,C 180,E1 13473.877,E2 13473.877} C_VEL
LIN {X 0,Y 329.756,Z 474.273,A -85,B 0,C 180,E1 13471.226,E2 13471.226} C_VEL
LIN {X 0,Y 337.689,Z 485.812,A -85,B 0,C 180,E1 13468.044,E2 13468.044} C_VEL
LIN {X 0,Y 345.954,Z 498.797,A -85,B 0,C 180,E1 13465.145,E2 13465.145} C_VEL
LIN {X 0,Y 347.77,Z 502.171,A -85,B 0,C 180,E1 13464.539,E2 13464.539} C_VEL
LIN {X 0,Y 337.342,Z 674.162,A -85,B 0,C 180,E1 13461.046,E2 13461.046} C_VEL
LIN {X 0,Y 335.352,Z 695.718,A -85,B 0,C 180,E1 13460.332,E2 13460.332} C_VEL
LIN {X 0,Y 332.466,Z 715.817,A -85,B 0,C 180,E1 13459.401,E2 13459.401} C_VEL
LIN {X 0,Y 328.765,Z 735.025,A -85,B 0,C 180,E1 13458.238,E2 13458.238} C_VEL
LIN {X 0,Y 324.089,Z 754.014,A -85,B 0,C 180,E1 13456.772,E2 13456.772} C_VEL
LIN {X 0,Y 318.707,Z 772.24,A -85,B 0,C 180,E1 13455.021,E2 13455.021} C_VEL
LIN {X 0,Y 312.633,Z 789.971,A -85,B 0,C 180,E1 13452.913,E2 13452.913} C_VEL
LIN {X 0,Y 306.505,Z 805.845,A -85,B 0,C 180,E1 13450.596,E2 13450.596} C_VEL
LIN {X 0,Y 300.306,Z 820.355,A -85,B 0,C 180,E1 13448.016,E2 13448.016} C_VEL
LIN {X 0,Y 294.028,Z 833.816,A -85,B 0,C 180,E1 13445.073,E2 13445.073} C_VEL
LIN {X 0,Y 288.071,Z 845.892,A -85,B 0,C 180,E1 13441.837,E2 13441.837} C_VEL
LIN {X 0,Y 282.405,Z 856.951,A -85,B 0,C 180,E1 13438.165,E2 13438.165} C_VEL
LIN {X 0,Y 277.639,Z 866.154,A -85,B 0,C 180,E1 13434.338,E2 13434.338} C_VEL
LIN {X 0,Y 273.502,Z 874.236,A -85,B 0,C 180,E1 13430.026,E2 13430.026} C_VEL
LIN {X 0,Y 270.467,Z 880.354,A -85,B 0,C 180,E1 13425.654,E2 13425.654} C_VEL
LIN {X 0,Y 268.445,Z 884.84,A -85,B 0,C 180,E1 13421.166,E2 13421.166} C_VEL
LIN {X 0,Y 267.229,Z 887.852,A -85,B 0,C 180,E1 13416.443,E2 13416.443} C_VEL
LIN {X 0,Y 266.752,Z 889.223,A -85,B 0,C 180,E1 13411.932,E2 13411.932} C_VEL
LIN {X 0,Y 266.795,Z 889.178,A -85,B 0,C 180,E1 13407.422,E2 13407.422} C_VEL
LIN {X 0,Y 267.335,Z 887.615,A -85,B 0,C 180,E1 13402.91,E2 13402.91} C_VEL
LIN {X 0,Y 268.568,Z 884.578,A -85,B 0,C 180,E1 13398.403,E2 13398.403} C_VEL
LIN {X 0,Y 270.792,Z 879.687,A -85,B 0,C 180,E1 13393.704,E2 13393.704} C_VEL
LIN {X 0,Y 273.834,Z 873.59,A -85,B 0,C 180,E1 13389.482,E2 13389.482} C_VEL
LIN {X 0,Y 277.919,Z 865.725,A -85,B 0,C 180,E1 13385.336,E2 13385.336} C_VEL
LIN {X 0,Y 282.782,Z 856.343,A -85,B 0,C 180,E1 13381.491,E2 13381.491} C_VEL
LIN {X 0,Y 288.295,Z 845.57,A -85,B 0,C 180,E1 13377.955,E2 13377.955} C_VEL
LIN {X 0,Y 294.677,Z 832.577,A -85,B 0,C 180,E1 13374.522,E2 13374.522} C_VEL
LIN {X 0,Y 301,Z 818.912,A -85,B 0,C 180,E1 13371.602,E2 13371.602} C_VEL
LIN {X 0,Y 307.323,Z 804.1,A -85,B 0,C 180,E1 13369.009,E2 13369.009} C_VEL
LIN {X 0,Y 313.485,Z 787.935,A -85,B 0,C 180,E1 13366.711,E2 13366.711} C_VEL
LIN {X 0,Y 319.144,Z 771.161,A -85,B 0,C 180,E1 13364.759,E2 13364.759} C_VEL
LIN {X 0,Y 324.602,Z 752.409,A -85,B 0,C 180,E1 13362.988,E2 13362.988} C_VEL
LIN {X 0,Y 328.984,Z 734.435,A -85,B 0,C 180,E1 13361.618,E2 13361.618} C_VEL
LIN {X 0,Y 332.717,Z 714.982,A -85,B 0,C 180,E1 13360.449,E2 13360.449} C_VEL
LIN {X 0,Y 333.007,Z 713.325,A -85,B 0,C 180,E1 13360.358,E2 13360.358} C_VEL
LIN {X 0,Y 333.498,Z 706.11,A -85,B 0,C 180,E1 13359.868,E2 13359.868} C_VEL
LIN {X 0,Y 332.263,Z 688.228,A -85,B 0,C 180,E1 13358.304,E2 13358.304} C_VEL
LIN {X 0,Y 332.375,Z 680.832,A -85,B 0,C 180,E1 13357.915,E2 13357.915} C_VEL
LIN {X 0,Y 334.388,Z 647.778,A -85,B 0,C 180,E1 13357.142,E2 13357.142} C_VEL
LIN {X 0,Y 343.393,Z 506.025,A -85,B 0,C 180,E1 13354.293,E2 13354.293} C_VEL
LIN {X 0,Y 335.188,Z 492.774,A -85,B 0,C 180,E1 13351.318,E2 13351.318} C_VEL
LIN {X 0,Y 328.079,Z 482.293,A -85,B 0,C 180,E1 13348.388,E2 13348.388} C_VEL
LIN {X 0,Y 322.689,Z 474.841,A -85,B 0,C 180,E1 13345.857,E2 13345.857} C_VEL
LIN {X 0,Y 319.364,Z 470.418,A -85,B 0,C 180,E1 13344.115,E2 13344.115} C_VEL
LIN {X 0,Y 316.234,Z 466.316,A -85,B 0,C 180,E1 13342.298,E2 13342.298} C_VEL
LIN {X 0,Y 312.244,Z 461.287,A -85,B 0,C 180,E1 13339.648,E2 13339.648} C_VEL
LIN {X 0,Y 308.031,Z 456.152,A -85,B 0,C 180,E1 13336.21,E2 13336.21} C_VEL
LIN {X 0,Y 303.027,Z 450.526,A -85,B 0,C 180,E1 13330.072,E2 13330.072} C_VEL
LIN {X 0,Y 301.133,Z 449.337,A -85,B 0,C 180,E1 13324.762,E2 13324.762} C_VEL
LIN {X 0,Y 301.596,Z 450.183,A -85,B 0,C 180,E1 13319.431,E2 13319.431} C_VEL
LIN {X 0,Y 305.162,Z 455.827,A -85,B 0,C 180,E1 13312.943,E2 13312.943} C_VEL
LIN {X 0,Y 309.041,Z 461.644,A -85,B 0,C 180,E1 13308.996,E2 13308.996} C_VEL
LIN {X 0,Y 312.367,Z 466.43,A -85,B 0,C 180,E1 13306.393,E2 13306.393} C_VEL
LIN {X 0,Y 316.93,Z 473.221,A -85,B 0,C 180,E1 13303.411,E2 13303.411} C_VEL
LIN {X 0,Y 322.515,Z 481.698,A -85,B 0,C 180,E1 13300.345,E2 13300.345} C_VEL
LIN {X 0,Y 329.27,Z 492.522,A -85,B 0,C 180,E1 13297.175,E2 13297.175} C_VEL
LIN {X 0,Y 336.943,Z 505.786,A -85,B 0,C 180,E1 13294.043,E2 13294.043} C_VEL
LIN {X 0,Y 344.548,Z 520.311,A -85,B 0,C 180,E1 13291.274,E2 13291.274} C_VEL
LIN {X 0,Y 344.675,Z 521.435,A -85,B 0,C 180,E1 13291.195,E2 13291.195} C_VEL
LIN {X 0,Y 330.42,Z 725.992,A -85,B 0,C 180,E1 13286.799,E2 13286.799} C_VEL
LIN {X 0,Y 327.597,Z 748.566,A -85,B 0,C 180,E1 13286.127,E2 13286.127} C_VEL
LIN {X 0,Y 323.462,Z 770.701,A -85,B 0,C 180,E1 13285.255,E2 13285.255} C_VEL
LIN {X 0,Y 318.654,Z 790.974,A -85,B 0,C 180,E1 13284.205,E2 13284.205} C_VEL
LIN {X 0,Y 312.994,Z 811,A -85,B 0,C 180,E1 13282.841,E2 13282.841} C_VEL
LIN {X 0,Y 306.486,Z 831.382,A -85,B 0,C 180,E1 13281.078,E2 13281.078} C_VEL
LIN {X 0,Y 299.837,Z 850.235,A -85,B 0,C 180,E1 13279.046,E2 13279.046} C_VEL
LIN {X 0,Y 292.877,Z 868.35,A -85,B 0,C 180,E1 13276.644,E2 13276.644} C_VEL
LIN {X 0,Y 285.909,Z 885.612,A -85,B 0,C 180,E1 13273.818,E2 13273.818} C_VEL
LIN {X 0,Y 279.251,Z 901.701,A -85,B 0,C 180,E1 13270.619,E2 13270.619} C_VEL
LIN {X 0,Y 273.188,Z 916.451,A -85,B 0,C 180,E1 13267.074,E2 13267.074} C_VEL
LIN {X 0,Y 267.766,Z 930.233,A -85,B 0,C 180,E1 13263.034,E2 13263.034} C_VEL
LIN {X 0,Y 263.477,Z 942.162,A -85,B 0,C 180,E1 13258.765,E2 13258.765} C_VEL
LIN {X 0,Y 260.226,Z 952.979,A -85,B 0,C 180,E1 13254.032,E2 13254.032} C_VEL
LIN {X 0,Y 258.361,Z 961.469,A -85,B 0,C 180,E1 13249.439,E2 13249.439} C_VEL
LIN {X 0,Y 257.557,Z 967.794,A -85,B 0,C 180,E1 13245.075,E2 13245.075} C_VEL
LIN {X 0,Y 257.494,Z 972.804,A -85,B 0,C 180,E1 13240.515,E2 13240.515} C_VEL
LIN {X 0,Y 257.772,Z 975.691,A -85,B 0,C 180,E1 13236.682,E2 13236.682} C_VEL
LIN {X 0,Y 258.098,Z 977.388,A -85,B 0,C 180,E1 13232.887,E2 13232.887} C_VEL
LIN {X 0,Y 258.191,Z 977.677,A -85,B 0,C 180,E1 13229.113,E2 13229.113} C_VEL
LIN {X 0,Y 257.991,Z 976.801,A -85,B 0,C 180,E1 13225.556,E2 13225.556} C_VEL
LIN {X 0,Y 257.606,Z 974.532,A -85,B 0,C 180,E1 13221.52,E2 13221.52} C_VEL
LIN {X 0,Y 257.456,Z 970.49,A -85,B 0,C 180,E1 13217.213,E2 13217.213} C_VEL
LIN {X 0,Y 257.903,Z 964.448,A -85,B 0,C 180,E1 13212.497,E2 13212.497} C_VEL
LIN {X 0,Y 259.246,Z 957.012,A -85,B 0,C 180,E1 13208.034,E2 13208.034} C_VEL
LIN {X 0,Y 261.765,Z 947.493,A -85,B 0,C 180,E1 13203.459,E2 13203.459} C_VEL
LIN {X 0,Y 265.584,Z 936.023,A -85,B 0,C 180,E1 13198.955,E2 13198.955} C_VEL
LIN {X 0,Y 270.495,Z 923.111,A -85,B 0,C 180,E1 13194.791,E2 13194.791} C_VEL
LIN {X 0,Y 276.341,Z 908.672,A -85,B 0,C 180,E1 13190.987,E2 13190.987} C_VEL
LIN {X 0,Y 282.623,Z 893.447,A -85,B 0,C 180,E1 13187.679,E2 13187.679} C_VEL
LIN {X 0,Y 289.752,Z 876.006,A -85,B 0,C 180,E1 13184.561,E2 13184.561} C_VEL
LIN {X 0,Y 296.657,Z 858.523,A -85,B 0,C 180,E1 13182.005,E2 13182.005} C_VEL
LIN {X 0,Y 303.632,Z 839.476,A -85,B 0,C 180,E1 13179.752,E2 13179.752} C_VEL
LIN {X 0,Y 309.976,Z 820.525,A -85,B 0,C 180,E1 13177.948,E2 13177.948} C_VEL
LIN {X 0,Y 316.086,Z 800.092,A -85,B 0,C 180,E1 13176.394,E2 13176.394} C_VEL
LIN {X 0,Y 321.406,Z 779.625,A -85,B 0,C 180,E1 13175.185,E2 13175.185} C_VEL
LIN {X 0,Y 326.001,Z 757.601,A -85,B 0,C 180,E1 13174.213,E2 13174.213} C_VEL
LIN {X 0,Y 329.315,Z 735.378,A -85,B 0,C 180,E1 13173.468,E2 13173.468} C_VEL
LIN {X 0,Y 331.723,Z 707.462,A -85,B 0,C 180,E1 13172.789,E2 13172.789} C_VEL
LIN {X 0,Y 344.608,Z 520.554,A -85,B 0,C 180,E1 13168.792,E2 13168.792} C_VEL
LIN {X 0,Y 336.921,Z 505.866,A -85,B 0,C 180,E1 13166.006,E2 13166.006} C_VEL
LIN {X 0,Y 329.232,Z 492.56,A -85,B 0,C 180,E1 13162.875,E2 13162.875} C_VEL
LIN {X 0,Y 322.47,Z 481.682,A -85,B 0,C 180,E1 13159.705,E2 13159.705} C_VEL
LIN {X 0,Y 316.798,Z 473.053,A -85,B 0,C 180,E1 13156.596,E2 13156.596} C_VEL
LIN {X 0,Y 313.477,Z 468.269,A -85,B 0,C 180,E1 13154.5,E2 13154.5} C_VEL
LIN {X 0,Y 311.131,Z 464.64,A -85,B 0,C 180,E1 13152.811,E2 13152.811} C_VEL
LIN {X 0,Y 307.855,Z 460.003,A -85,B 0,C 180,E1 13150.1,E2 13150.1} C_VEL
LIN {X 0,Y 304.608,Z 455.025,A -85,B 0,C 180,E1 13146.597,E2 13146.597} C_VEL
LIN {X 0,Y 301.366,Z 449.989,A -85,B 0,C 180,E1 13140.57,E2 13140.57} C_VEL
LIN {X 0,Y 300.957,Z 449.166,A -85,B 0,C 180,E1 13134.662,E2 13134.662} C_VEL
LIN {X 0,Y 303.074,Z 450.54,A -85,B 0,C 180,E1 13129.353,E2 13129.353} C_VEL
LIN {X 0,Y 308.742,Z 457.003,A -85,B 0,C 180,E1 13122.86,E2 13122.86} C_VEL
LIN {X 0,Y 313.341,Z 462.67,A -85,B 0,C 180,E1 13119.353,E2 13119.353} C_VEL
LIN {X 0,Y 317.776,Z 468.317,A -85,B 0,C 180,E1 13116.594,E2 13116.594} C_VEL
LIN {X 0,Y 322.136,Z 474.161,A -85,B 0,C 180,E1 13114.244,E2 13114.244} C_VEL
LIN {X 0,Y 327.594,Z 481.615,A -85,B 0,C 180,E1 13111.666,E2 13111.666} C_VEL
LIN {X 0,Y 335.182,Z 492.867,A -85,B 0,C 180,E1 13108.531,E2 13108.531} C_VEL
LIN {X 0,Y 343.305,Z 505.976,A -85,B 0,C 180,E1 13105.596,E2 13105.596} C_VEL
LIN {X 0,Y 332.645,Z 675.109,A -85,B 0,C 180,E1 13102.142,E2 13102.142} C_VEL
LIN {X 0,Y 330.582,Z 696.653,A -85,B 0,C 180,E1 13101.426,E2 13101.426} C_VEL
LIN {X 0,Y 327.563,Z 716.955,A -85,B 0,C 180,E1 13100.481,E2 13100.481} C_VEL
LIN {X 0,Y 323.712,Z 736.254,A -85,B 0,C 180,E1 13099.305,E2 13099.305} C_VEL
LIN {X 0,Y 319.022,Z 754.682,A -85,B 0,C 180,E1 13097.878,E2 13097.878} C_VEL
LIN {X 0,Y 313.46,Z 772.977,A -85,B 0,C 180,E1 13096.121,E2 13096.121} C_VEL
LIN {X 0,Y 307.449,Z 790.053,A -85,B 0,C 180,E1 13094.097,E2 13094.097} C_VEL
LIN {X 0,Y 301.025,Z 806.21,A -85,B 0,C 180,E1 13091.75,E2 13091.75} C_VEL
LIN {X 0,Y 294.554,Z 820.802,A -85,B 0,C 180,E1 13089.146,E2 13089.146} C_VEL
LIN {X 0,Y 287.975,Z 834.405,A -85,B 0,C 180,E1 13086.169,E2 13086.169} C_VEL
LIN {X 0,Y 281.721,Z 846.605,A -85,B 0,C 180,E1 13082.884,E2 13082.884} C_VEL
LIN {X 0,Y 275.931,Z 857.428,A -85,B 0,C 180,E1 13079.283,E2 13079.283} C_VEL
LIN {X 0,Y 270.805,Z 866.845,A -85,B 0,C 180,E1 13075.356,E2 13075.356} C_VEL
LIN {X 0,Y 266.467,Z 874.744,A -85,B 0,C 180,E1 13071.111,E2 13071.111} C_VEL
LIN {X 0,Y 263.229,Z 880.885,A -85,B 0,C 180,E1 13066.776,E2 13066.776} C_VEL
LIN {X 0,Y 260.835,Z 885.814,A -85,B 0,C 180,E1 13061.944,E2 13061.944} C_VEL
LIN {X 0,Y 259.511,Z 888.889,A -85,B 0,C 180,E1 13057.303,E2 13057.303} C_VEL
LIN {X 0,Y 258.92,Z 890.484,A -85,B 0,C 180,E1 13052.655,E2 13052.655} C_VEL
LIN {X 0,Y 258.851,Z 890.581,A -85,B 0,C 180,E1 13048.229,E2 13048.229} C_VEL
LIN {X 0,Y 259.329,Z 889.336,A -85,B 0,C 180,E1 13043.58,E2 13043.58} C_VEL
LIN {X 0,Y 260.506,Z 886.636,A -85,B 0,C 180,E1 13038.936,E2 13038.936} C_VEL
LIN {X 0,Y 262.548,Z 882.356,A -85,B 0,C 180,E1 13034.313,E2 13034.313} C_VEL
LIN {X 0,Y 265.691,Z 876.284,A -85,B 0,C 180,E1 13029.745,E2 13029.745} C_VEL
LIN {X 0,Y 269.759,Z 868.742,A -85,B 0,C 180,E1 13025.475,E2 13025.475} C_VEL
LIN {X 0,Y 274.956,Z 859.277,A -85,B 0,C 180,E1 13021.316,E2 13021.316} C_VEL
LIN {X 0,Y 280.845,Z 848.388,A -85,B 0,C 180,E1 13017.54,E2 13017.54} C_VEL
LIN {X 0,Y 287.096,Z 836.38,A -85,B 0,C 180,E1 13014.194,E2 13014.194} C_VEL
LIN {X 0,Y 293.999,Z 822.209,A -85,B 0,C 180,E1 13011.015,E2 13011.015} C_VEL
LIN {X 0,Y 300.657,Z 807.246,A -85,B 0,C 180,E1 13008.313,E2 13008.313} C_VEL
LIN {X 0,Y 306.816,Z 791.94,A -85,B 0,C 180,E1 13006.047,E2 13006.047} C_VEL
LIN {X 0,Y 313.065,Z 774.489,A -85,B 0,C 180,E1 13003.935,E2 13003.935} C_VEL
LIN {X 0,Y 318.54,Z 756.866,A -85,B 0,C 180,E1 13002.201,E2 13002.201} C_VEL
LIN {X 0,Y 323.343,Z 738.21,A -85,B 0,C 180,E1 13000.728,E2 13000.728} C_VEL
LIN {X 0,Y 327.294,Z 718.997,A -85,B 0,C 180,E1 12999.529,E2 12999.529} C_VEL
LIN {X 0,Y 330.519,Z 698.051,A -85,B 0,C 180,E1 12998.527,E2 12998.527} C_VEL
LIN {X 0,Y 332.375,Z 680.832,A -85,B 0,C 180,E1 12997.915,E2 12997.915} C_VEL
LIN {X 0,Y 332.44,Z 673.352,A -85,B 0,C 180,E1 12997.554,E2 12997.554} C_VEL
LIN {X 0,Y 330.015,Z 653.734,A -85,B 0,C 180,E1 12996.217,E2 12996.217} C_VEL
LIN {X 0,Y 329.984,Z 647.235,A -85,B 0,C 180,E1 12995.98,E2 12995.98} C_VEL
LIN {X 0,Y 339.029,Z 510.242,A -85,B 0,C 180,E1 12993.217,E2 12993.217} C_VEL
LIN {X 0,Y 331.824,Z 498.478,A -85,B 0,C 180,E1 12990.468,E2 12990.468} C_VEL
LIN {X 0,Y 324.775,Z 487.833,A -85,B 0,C 180,E1 12987.404,E2 12987.404} C_VEL
LIN {X 0,Y 318.433,Z 478.928,A -85,B 0,C 180,E1 12984.19,E2 12984.19} C_VEL
LIN {X 0,Y 314.435,Z 473.725,A -85,B 0,C 180,E1 12981.842,E2 12981.842} C_VEL
LIN {X 0,Y 310.68,Z 468.87,A -85,B 0,C 180,E1 12979.262,E2 12979.262} C_VEL
LIN {X 0,Y 306.739,Z 463.935,A -85,B 0,C 180,E1 12975.949,E2 12975.949} C_VEL
LIN {X 0,Y 301.955,Z 458.418,A -85,B 0,C 180,E1 12969.915,E2 12969.915} C_VEL
LIN {X 0,Y 300.162,Z 457.278,A -85,B 0,C 180,E1 12964.777,E2 12964.777} C_VEL
LIN {X 0,Y 300.564,Z 458.062,A -85,B 0,C 180,E1 12959.619,E2 12959.619} C_VEL
LIN {X 0,Y 303.872,Z 463.511,A -85,B 0,C 180,E1 12953.292,E2 12953.292} C_VEL
LIN {X 0,Y 307.525,Z 469.169,A -85,B 0,C 180,E1 12949.415,E2 12949.415} C_VEL
LIN {X 0,Y 310.743,Z 473.979,A -85,B 0,C 180,E1 12946.794,E2 12946.794} C_VEL
LIN {X 0,Y 315.188,Z 480.77,A -85,B 0,C 180,E1 12943.79,E2 12943.79} C_VEL
LIN {X 0,Y 320.653,Z 489.325,A -85,B 0,C 180,E1 12940.7,E2 12940.7} C_VEL
LIN {X 0,Y 327.374,Z 500.453,A -85,B 0,C 180,E1 12937.462,E2 12937.462} C_VEL
LIN {X 0,Y 334.808,Z 513.819,A -85,B 0,C 180,E1 12934.341,E2 12934.341} C_VEL
LIN {X 0,Y 340.249,Z 524.705,A -85,B 0,C 180,E1 12932.271,E2 12932.271} C_VEL
LIN {X 0,Y 325.758,Z 725.67,A -85,B 0,C 180,E1 12927.942,E2 12927.942} C_VEL
LIN {X 0,Y 322.875,Z 747.824,A -85,B 0,C 180,E1 12927.278,E2 12927.278} C_VEL
LIN {X 0,Y 318.5,Z 770.465,A -85,B 0,C 180,E1 12926.381,E2 12926.381} C_VEL
LIN {X 0,Y 313.254,Z 791.658,A -85,B 0,C 180,E1 12925.268,E2 12925.268} C_VEL
LIN {X 0,Y 307.459,Z 811.388,A -85,B 0,C 180,E1 12923.906,E2 12923.906} C_VEL
LIN {X 0,Y 301.047,Z 830.629,A -85,B 0,C 180,E1 12922.222,E2 12922.222} C_VEL
LIN {X 0,Y 293.883,Z 850.097,A -85,B 0,C 180,E1 12920.098,E2 12920.098} C_VEL
LIN {X 0,Y 286.685,Z 868.105,A -85,B 0,C 180,E1 12917.674,E2 12917.674} C_VEL
LIN {X 0,Y 279.438,Z 885.197,A -85,B 0,C 180,E1 12914.816,E2 12914.816} C_VEL
LIN {X 0,Y 272.383,Z 901.393,A -85,B 0,C 180,E1 12911.511,E2 12911.511} C_VEL
LIN {X 0,Y 265.901,Z 916.32,A -85,B 0,C 180,E1 12907.798,E2 12907.798} C_VEL
LIN {X 0,Y 260.447,Z 929.481,A -85,B 0,C 180,E1 12903.822,E2 12903.822} C_VEL
LIN {X 0,Y 255.854,Z 941.477,A -85,B 0,C 180,E1 12899.372,E2 12899.372} C_VEL
LIN {X 0,Y 252.463,Z 952.024,A -85,B 0,C 180,E1 12894.571,E2 12894.571} C_VEL
LIN {X 0,Y 250.476,Z 960.425,A -85,B 0,C 180,E1 12889.833,E2 12889.833} C_VEL
LIN {X 0,Y 249.623,Z 966.712,A -85,B 0,C 180,E1 12885.328,E2 12885.328} C_VEL
LIN {X 0,Y 249.555,Z 971.639,A -85,B 0,C 180,E1 12880.62,E2 12880.62} C_VEL
LIN {X 0,Y 249.883,Z 974.625,A -85,B 0,C 180,E1 12876.433,E2 12876.433} C_VEL
LIN {X 0,Y 250.225,Z 976.138,A -85,B 0,C 180,E1 12872.52,E2 12872.52} C_VEL
LIN {X 0,Y 250.299,Z 976.321,A -85,B 0,C 180,E1 12868.856,E2 12868.856} C_VEL
LIN {X 0,Y 250.08,Z 975.465,A -85,B 0,C 180,E1 12865.415,E2 12865.415} C_VEL
LIN {X 0,Y 249.657,Z 973.177,A -85,B 0,C 180,E1 12861.248,E2 12861.248} C_VEL
LIN {X 0,Y 249.516,Z 969.114,A -85,B 0,C 180,E1 12856.799,E2 12856.799} C_VEL
LIN {X 0,Y 250.002,Z 963.257,A -85,B 0,C 180,E1 12852.067,E2 12852.067} C_VEL
LIN {X 0,Y 251.526,Z 955.598,A -85,B 0,C 180,E1 12847.323,E2 12847.323} C_VEL
LIN {X 0,Y 254.275,Z 946.061,A -85,B 0,C 180,E1 12842.613,E2 12842.613} C_VEL
LIN {X 0,Y 258.486,Z 934.319,A -85,B 0,C 180,E1 12837.899,E2 12837.899} C_VEL
LIN {X 0,Y 263.633,Z 921.647,A -85,B 0,C 180,E1 12833.731,E2 12833.731} C_VEL
LIN {X 0,Y 269.816,Z 907.199,A -85,B 0,C 180,E1 12829.856,E2 12829.856} C_VEL
LIN {X 0,Y 276.528,Z 891.793,A -85,B 0,C 180,E1 12826.471,E2 12826.471} C_VEL
LIN {X 0,Y 284.161,Z 873.902,A -85,B 0,C 180,E1 12823.258,E2 12823.258} C_VEL
LIN {X 0,Y 291.428,Z 856.184,A -85,B 0,C 180,E1 12820.682,E2 12820.682} C_VEL
LIN {X 0,Y 298.688,Z 837.138,A -85,B 0,C 180,E1 12818.443,E2 12818.443} C_VEL
LIN {X 0,Y 305.276,Z 817.951,A -85,B 0,C 180,E1 12816.645,E2 12816.645} C_VEL
LIN {X 0,Y 311.607,Z 797.18,A -85,B 0,C 180,E1 12815.102,E2 12815.102} C_VEL
LIN {X 0,Y 316.937,Z 776.983,A -85,B 0,C 180,E1 12813.942,E2 12813.942} C_VEL
LIN {X 0,Y 321.591,Z 754.977,A -85,B 0,C 180,E1 12812.989,E2 12812.989} C_VEL
LIN {X 0,Y 324.852,Z 732.964,A -85,B 0,C 180,E1 12812.269,E2 12812.269} C_VEL
LIN {X 0,Y 327.403,Z 703.005,A -85,B 0,C 180,E1 12811.555,E2 12811.555} C_VEL
LIN {X 0,Y 340.135,Z 524.352,A -85,B 0,C 180,E1 12807.727,E2 12807.727} C_VEL
LIN {X 0,Y 332.999,Z 510.638,A -85,B 0,C 180,E1 12804.999,E2 12804.999} C_VEL
LIN {X 0,Y 326.057,Z 498.335,A -85,B 0,C 180,E1 12802.016,E2 12802.016} C_VEL
LIN {X 0,Y 318.776,Z 486.316,A -85,B 0,C 180,E1 12798.374,E2 12798.374} C_VEL
LIN {X 0,Y 313.137,Z 477.585,A -85,B 0,C 180,E1 12794.989,E2 12794.989} C_VEL
LIN {X 0,Y 309.303,Z 471.886,A -85,B 0,C 180,E1 12792.224,E2 12792.224} C_VEL
LIN {X 0,Y 306.368,Z 467.566,A -85,B 0,C 180,E1 12789.675,E2 12789.675} C_VEL
LIN {X 0,Y 303.327,Z 462.746,A -85,B 0,C 180,E1 12786.244,E2 12786.244} C_VEL
LIN {X 0,Y 300.331,Z 457.881,A -85,B 0,C 180,E1 12780.381,E2 12780.381} C_VEL
LIN {X 0,Y 299.986,Z 457.109,A -85,B 0,C 180,E1 12774.645,E2 12774.645} C_VEL
LIN {X 0,Y 302.109,Z 458.541,A -85,B 0,C 180,E1 12769.319,E2 12769.319} C_VEL
LIN {X 0,Y 307.372,Z 464.732,A -85,B 0,C 180,E1 12763.171,E2 12763.171} C_VEL
LIN {X 0,Y 311.745,Z 470.253,A -85,B 0,C 180,E1 12759.733,E2 12759.733} C_VEL
LIN {X 0,Y 316.008,Z 475.814,A -85,B 0,C 180,E1 12756.998,E2 12756.998} C_VEL
LIN {X 0,Y 320.357,Z 481.781,A -85,B 0,C 180,E1 12754.586,E2 12754.586} C_VEL
LIN {X 0,Y 325.81,Z 489.513,A -85,B 0,C 180,E1 12751.946,E2 12751.946} C_VEL
LIN {X 0,Y 333.108,Z 500.533,A -85,B 0,C 180,E1 12748.867,E2 12748.867} C_VEL
LIN {X 0,Y 338.932,Z 510.316,A -85,B 0,C 180,E1 12746.668,E2 12746.668} C_VEL
LIN {X 0,Y 328.094,Z 675.74,A -85,B 0,C 180,E1 12743.279,E2 12743.279} C_VEL
LIN {X 0,Y 325.93,Z 697.638,A -85,B 0,C 180,E1 12742.549,E2 12742.549} C_VEL
LIN {X 0,Y 322.918,Z 717.367,A -85,B 0,C 180,E1 12741.633,E2 12741.633} C_VEL
LIN {X 0,Y 318.934,Z 736.763,A -85,B 0,C 180,E1 12740.455,E2 12740.455} C_VEL
LIN {X 0,Y 314.077,Z 755.35,A -85,B 0,C 180,E1 12739.019,E2 12739.019} C_VEL
LIN {X 0,Y 308.334,Z 773.712,A -85,B 0,C 180,E1 12737.257,E2 12737.257} C_VEL
LIN {X 0,Y 302.104,Z 790.869,A -85,B 0,C 180,E1 12735.222,E2 12735.222} C_VEL
LIN {X 0,Y 295.431,Z 807.098,A -85,B 0,C 180,E1 12732.858,E2 12732.858} C_VEL
LIN {X 0,Y 288.475,Z 822.205,A -85,B 0,C 180,E1 12730.136,E2 12730.136} C_VEL
LIN {X 0,Y 281.629,Z 835.787,A -85,B 0,C 180,E1 12727.119,E2 12727.119} C_VEL
LIN {X 0,Y 275.103,Z 847.969,A -85,B 0,C 180,E1 12723.78,E2 12723.78} C_VEL
LIN {X 0,Y 269.039,Z 858.781,A -85,B 0,C 180,E1 12720.109,E2 12720.109} C_VEL
LIN {X 0,Y 263.654,Z 868.195,A -85,B 0,C 180,E1 12716.094,E2 12716.094} C_VEL
LIN {X 0,Y 258.882,Z 876.456,A -85,B 0,C 180,E1 12711.522,E2 12711.522} C_VEL
LIN {X 0,Y 255.501,Z 882.496,A -85,B 0,C 180,E1 12707.065,E2 12707.065} C_VEL
LIN {X 0,Y 253.088,Z 887.15,A -85,B 0,C 180,E1 12702.316,E2 12702.316} C_VEL
LIN {X 0,Y 251.673,Z 890.22,A -85,B 0,C 180,E1 12697.532,E2 12697.532} C_VEL
LIN {X 0,Y 251.037,Z 891.813,A -85,B 0,C 180,E1 12692.738,E2 12692.738} C_VEL
LIN {X 0,Y 250.964,Z 891.909,A -85,B 0,C 180,E1 12688.173,E2 12688.173} C_VEL
LIN {X 0,Y 251.477,Z 890.667,A -85,B 0,C 180,E1 12683.379,E2 12683.379} C_VEL
LIN {X 0,Y 252.737,Z 887.971,A -85,B 0,C 180,E1 12678.592,E2 12678.592} C_VEL
LIN {X 0,Y 254.919,Z 883.692,A -85,B 0,C 180,E1 12673.831,E2 12673.831} C_VEL
LIN {X 0,Y 258.253,Z 877.625,A -85,B 0,C 180,E1 12669.135,E2 12669.135} C_VEL
LIN {X 0,Y 262.557,Z 870.087,A -85,B 0,C 180,E1 12664.755,E2 12664.755} C_VEL
LIN {X 0,Y 268.022,Z 860.63,A -85,B 0,C 180,E1 12660.502,E2 12660.502} C_VEL
LIN {X 0,Y 273.923,Z 850.247,A -85,B 0,C 180,E1 12656.806,E2 12656.806} C_VEL
LIN {X 0,Y 280.321,Z 838.529,A -85,B 0,C 180,E1 12653.444,E2 12653.444} C_VEL
LIN {X 0,Y 287.291,Z 824.785,A -85,B 0,C 180,E1 12650.278,E2 12650.278} C_VEL
LIN {X 0,Y 293.864,Z 810.763,A -85,B 0,C 180,E1 12647.652,E2 12647.652} C_VEL
LIN {X 0,Y 300.696,Z 794.665,A -85,B 0,C 180,E1 12645.181,E2 12645.181} C_VEL
LIN {X 0,Y 307.016,Z 777.934,A -85,B 0,C 180,E1 12643.09,E2 12643.09} C_VEL
LIN {X 0,Y 313.038,Z 759.411,A -85,B 0,C 180,E1 12641.224,E2 12641.224} C_VEL
LIN {X 0,Y 317.954,Z 741.164,A -85,B 0,C 180,E1 12639.753,E2 12639.753} C_VEL
LIN {X 0,Y 322.233,Z 721.564,A -85,B 0,C 180,E1 12638.497,E2 12638.497} C_VEL
LIN {X 0,Y 325.531,Z 701.681,A -85,B 0,C 180,E1 12637.513,E2 12637.513} C_VEL
LIN {X 0,Y 327.852,Z 681.194,A -85,B 0,C 180,E1 12636.769,E2 12636.769} C_VEL
LIN {X 0,Y 329.984,Z 647.235,A -85,B 0,C 180,E1 12635.98,E2 12635.98} C_VEL
LIN {X 0,Y 329.937,Z 639.66,A -85,B 0,C 180,E1 12635.683,E2 12635.683} C_VEL
LIN {X 0,Y 327.913,Z 619.921,A -85,B 0,C 180,E1 12634.356,E2 12634.356} C_VEL
LIN {X 0,Y 327.968,Z 613.408,A -85,B 0,C 180,E1 12634.113,E2 12634.113} C_VEL
LIN {X 0,Y 334.787,Z 514.493,A -85,B 0,C 180,E1 12632.114,E2 12632.114} C_VEL
LIN {X 0,Y 327.838,Z 503.03,A -85,B 0,C 180,E1 12629.298,E2 12629.298} C_VEL
LIN {X 0,Y 321.041,Z 492.822,A -85,B 0,C 180,E1 12626.148,E2 12626.148} C_VEL
LIN {X 0,Y 315.792,Z 485.375,A -85,B 0,C 180,E1 12623.315,E2 12623.315} C_VEL
LIN {X 0,Y 312.659,Z 481.131,A -85,B 0,C 180,E1 12621.381,E2 12621.381} C_VEL
LIN {X 0,Y 309.12,Z 476.452,A -85,B 0,C 180,E1 12618.872,E2 12618.872} C_VEL
LIN {X 0,Y 305.53,Z 471.78,A -85,B 0,C 180,E1 12615.761,E2 12615.761} C_VEL
LIN {X 0,Y 300.885,Z 466.31,A -85,B 0,C 180,E1 12609.758,E2 12609.758} C_VEL
LIN {X 0,Y 299.19,Z 465.218,A -85,B 0,C 180,E1 12604.793,E2 12604.793} C_VEL
LIN {X 0,Y 299.584,Z 466.04,A -85,B 0,C 180,E1 12599.618,E2 12599.618} C_VEL
LIN {X 0,Y 302.659,Z 471.35,A -85,B 0,C 180,E1 12593.551,E2 12593.551} C_VEL
LIN {X 0,Y 306.121,Z 476.87,A -85,B 0,C 180,E1 12589.747,E2 12589.747} C_VEL
LIN {X 0,Y 309.139,Z 481.525,A -85,B 0,C 180,E1 12587.2,E2 12587.2} C_VEL
LIN {X 0,Y 313.541,Z 488.419,A -85,B 0,C 180,E1 12584.131,E2 12584.131} C_VEL
LIN {X 0,Y 318.976,Z 497.193,A -85,B 0,C 180,E1 12580.974,E2 12580.974} C_VEL
LIN {X 0,Y 326.003,Z 509.392,A -85,B 0,C 180,E1 12577.505,E2 12577.505} C_VEL
LIN {X 0,Y 332.872,Z 522.296,A -85,B 0,C 180,E1 12574.562,E2 12574.562} C_VEL
LIN {X 0,Y 335.889,Z 528.691,A -85,B 0,C 180,E1 12573.358,E2 12573.358} C_VEL
LIN {X 0,Y 321.257,Z 725.065,A -85,B 0,C 180,E1 12569.125,E2 12569.125} C_VEL
LIN {X 0,Y 318.294,Z 747.048,A -85,B 0,C 180,E1 12568.464,E2 12568.464} C_VEL
LIN {X 0,Y 313.667,Z 770.228,A -85,B 0,C 180,E1 12567.543,E2 12567.543} C_VEL
LIN {X 0,Y 308.318,Z 791.083,A -85,B 0,C 180,E1 12566.446,E2 12566.446} C_VEL
LIN {X 0,Y 302.033,Z 811.78,A -85,B 0,C 180,E1 12565.011,E2 12565.011} C_VEL
LIN {X 0,Y 295.126,Z 831.564,A -85,B 0,C 180,E1 12563.242,E2 12563.242} C_VEL
LIN {X 0,Y 287.748,Z 850.661,A -85,B 0,C 180,E1 12561.104,E2 12561.104} C_VEL
LIN {X 0,Y 280.32,Z 868.388,A -85,B 0,C 180,E1 12558.656,E2 12558.656} C_VEL
LIN {X 0,Y 272.584,Z 885.87,A -85,B 0,C 180,E1 12555.661,E2 12555.661} C_VEL
LIN {X 0,Y 265.463,Z 901.348,A -85,B 0,C 180,E1 12552.388,E2 12552.388} C_VEL
LIN {X 0,Y 258.562,Z 916.401,A -85,B 0,C 180,E1 12548.502,E2 12548.502} C_VEL
LIN {X 0,Y 252.894,Z 929.338,A -85,B 0,C 180,E1 12544.425,E2 12544.425} C_VEL
LIN {X 0,Y 248.007,Z 941.498,A -85,B 0,C 180,E1 12539.726,E2 12539.726} C_VEL
LIN {X 0,Y 244.585,Z 951.534,A -85,B 0,C 180,E1 12534.9,E2 12534.9} C_VEL
LIN {X 0,Y 242.46,Z 960.096,A -85,B 0,C 180,E1 12529.763,E2 12529.763} C_VEL
LIN {X 0,Y 241.611,Z 966.49,A -85,B 0,C 180,E1 12524.866,E2 12524.866} C_VEL
LIN {X 0,Y 241.643,Z 970.867,A -85,B 0,C 180,E1 12520.249,E2 12520.249} C_VEL
LIN {X 0,Y 242.064,Z 973.775,A -85,B 0,C 180,E1 12515.69,E2 12515.69} C_VEL
LIN {X 0,Y 242.373,Z 974.905,A -85,B 0,C 180,E1 12511.892,E2 12511.892} C_VEL
LIN {X 0,Y 242.4,Z 974.964,A -85,B 0,C 180,E1 12508.583,E2 12508.583} C_VEL
LIN {X 0,Y 242.12,Z 973.951,A -85,B 0,C 180,E1 12504.789,E2 12504.789} C_VEL
LIN {X 0,Y 241.674,Z 971.244,A -85,B 0,C 180,E1 12500.236,E2 12500.236} C_VEL
LIN {X 0,Y 241.573,Z 967.231,A -85,B 0,C 180,E1 12495.868,E2 12495.868} C_VEL
LIN {X 0,Y 242.33,Z 960.789,A -85,B 0,C 180,E1 12490.729,E2 12490.729} C_VEL
LIN {X 0,Y 244.196,Z 952.897,A -85,B 0,C 180,E1 12485.833,E2 12485.833} C_VEL
LIN {X 0,Y 247.402,Z 943.061,A -85,B 0,C 180,E1 12480.993,E2 12480.993} C_VEL
LIN {X 0,Y 251.794,Z 931.84,A -85,B 0,C 180,E1 12476.5,E2 12476.5} C_VEL
LIN {X 0,Y 257.53,Z 918.643,A -85,B 0,C 180,E1 12472.167,E2 12472.167} C_VEL
LIN {X 0,Y 264.223,Z 904.008,A -85,B 0,C 180,E1 12468.246,E2 12468.246} C_VEL
LIN {X 0,Y 271.515,Z 888.073,A -85,B 0,C 180,E1 12464.79,E2 12464.79} C_VEL
LIN {X 0,Y 278.992,Z 871.208,A -85,B 0,C 180,E1 12461.811,E2 12461.811} C_VEL
LIN {X 0,Y 286.881,Z 852.612,A -85,B 0,C 180,E1 12459.16,E2 12459.16} C_VEL
LIN {X 0,Y 294.205,Z 833.909,A -85,B 0,C 180,E1 12457.007,E2 12457.007} C_VEL
LIN {X 0,Y 301.057,Z 814.448,A -85,B 0,C 180,E1 12455.223,E2 12455.223} C_VEL
LIN {X 0,Y 307.258,Z 794.39,A -85,B 0,C 180,E1 12453.781,E2 12453.781} C_VEL
LIN {X 0,Y 312.963,Z 772.805,A -85,B 0,C 180,E1 12452.591,E2 12452.591} C_VEL
LIN {X 0,Y 317.501,Z 751.264,A -85,B 0,C 180,E1 12451.694,E2 12451.694} C_VEL
LIN {X 0,Y 320.777,Z 728.647,A -85,B 0,C 180,E1 12450.981,E2 12450.981} C_VEL
LIN {X 0,Y 324.47,Z 681.625,A -85,B 0,C 180,E1 12449.921,E2 12449.921} C_VEL
LIN {X 0,Y 335.751,Z 528.214,A -85,B 0,C 180,E1 12446.627,E2 12446.627} C_VEL
LIN {X 0,Y 328.904,Z 514.828,A -85,B 0,C 180,E1 12443.848,E2 12443.848} C_VEL
LIN {X 0,Y 323.035,Z 504.33,A -85,B 0,C 180,E1 12441.184,E2 12441.184} C_VEL
LIN {X 0,Y 316.57,Z 493.33,A -85,B 0,C 180,E1 12437.792,E2 12437.792} C_VEL
LIN {X 0,Y 311.185,Z 484.768,A -85,B 0,C 180,E1 12434.419,E2 12434.419} C_VEL
LIN {X 0,Y 307.726,Z 479.415,A -85,B 0,C 180,E1 12431.811,E2 12431.811} C_VEL
LIN {X 0,Y 304.89,Z 475.125,A -85,B 0,C 180,E1 12429.247,E2 12429.247} C_VEL
LIN {X 0,Y 302.055,Z 470.468,A -85,B 0,C 180,E1 12425.889,E2 12425.889} C_VEL
LIN {X 0,Y 299.298,Z 465.776,A -85,B 0,C 180,E1 12420.191,E2 12420.191} C_VEL
LIN {X 0,Y 299.018,Z 465.051,A -85,B 0,C 180,E1 12414.627,E2 12414.627} C_VEL
LIN {X 0,Y 301.036,Z 466.429,A -85,B 0,C 180,E1 12409.474,E2 12409.474} C_VEL
LIN {X 0,Y 306.011,Z 472.458,A -85,B 0,C 180,E1 12403.485,E2 12403.485} C_VEL
LIN {X 0,Y 310.284,Z 478.022,A -85,B 0,C 180,E1 12400.027,E2 12400.027} C_VEL
LIN {X 0,Y 314.324,Z 483.415,A -85,B 0,C 180,E1 12397.362,E2 12397.362} C_VEL
LIN {X 0,Y 318.592,Z 489.394,A -85,B 0,C 180,E1 12394.932,E2 12394.932} C_VEL
LIN {X 0,Y 324.486,Z 498.049,A -85,B 0,C 180,E1 12392.021,E2 12392.021} C_VEL
LIN {X 0,Y 331.036,Z 508.303,A -85,B 0,C 180,E1 12389.205,E2 12389.205} C_VEL
LIN {X 0,Y 334.665,Z 514.723,A -85,B 0,C 180,E1 12387.767,E2 12387.767} C_VEL
LIN {X 0,Y 323.664,Z 676.536,A -85,B 0,C 180,E1 12384.441,E2 12384.441} C_VEL
LIN {X 0,Y 321.422,Z 698.505,A -85,B 0,C 180,E1 12383.709,E2 12383.709} C_VEL
LIN {X 0,Y 318.265,Z 718.498,A -85,B 0,C 180,E1 12382.778,E2 12382.778} C_VEL
LIN {X 0,Y 314.008,Z 738.5,A -85,B 0,C 180,E1 12381.556,E2 12381.556} C_VEL
LIN {X 0,Y 308.898,Z 757.281,A -85,B 0,C 180,E1 12380.089,E2 12380.089} C_VEL
LIN {X 0,Y 303.057,Z 775.227,A -85,B 0,C 180,E1 12378.348,E2 12378.348} C_VEL
LIN {X 0,Y 296.518,Z 792.555,A -85,B 0,C 180,E1 12376.27,E2 12376.27} C_VEL
LIN {X 0,Y 289.702,Z 808.512,A -85,B 0,C 180,E1 12373.919,E2 12373.919} C_VEL
LIN {X 0,Y 282.486,Z 823.607,A -85,B 0,C 180,E1 12371.168,E2 12371.168} C_VEL
LIN {X 0,Y 275.363,Z 837.165,A -85,B 0,C 180,E1 12368.112,E2 12368.112} C_VEL
LIN {X 0,Y 268.556,Z 849.334,A -85,B 0,C 180,E1 12364.72,E2 12364.72} C_VEL
LIN {X 0,Y 262.206,Z 860.136,A -85,B 0,C 180,E1 12360.979,E2 12360.979} C_VEL
LIN {X 0,Y 256.375,Z 869.814,A -85,B 0,C 180,E1 12356.734,E2 12356.734} C_VEL
LIN {X 0,Y 251.429,Z 877.953,A -85,B 0,C 180,E1 12352.092,E2 12352.092} C_VEL
LIN {X 0,Y 247.779,Z 884.105,A -85,B 0,C 180,E1 12347.372,E2 12347.372} C_VEL
LIN {X 0,Y 245.26,Z 888.666,A -85,B 0,C 180,E1 12342.476,E2 12342.476} C_VEL
LIN {X 0,Y 243.733,Z 891.747,A -85,B 0,C 180,E1 12337.305,E2 12337.305} C_VEL
LIN {X 0,Y 243.115,Z 893.189,A -85,B 0,C 180,E1 12332.356,E2 12332.356} C_VEL
LIN {X 0,Y 243.109,Z 893.2,A -85,B 0,C 180,E1 12327.642,E2 12327.642} C_VEL
LIN {X 0,Y 243.717,Z 891.802,A -85,B 0,C 180,E1 12322.693,E2 12322.693} C_VEL
LIN {X 0,Y 245.232,Z 888.763,A -85,B 0,C 180,E1 12317.521,E2 12317.521} C_VEL
LIN {X 0,Y 247.735,Z 884.243,A -85,B 0,C 180,E1 12312.624,E2 12312.624} C_VEL
LIN {X 0,Y 251.452,Z 877.988,A -85,B 0,C 180,E1 12307.807,E2 12307.807} C_VEL
LIN {X 0,Y 256.466,Z 869.758,A -85,B 0,C 180,E1 12303.115,E2 12303.115} C_VEL
LIN {X 0,Y 262.108,Z 860.395,A -85,B 0,C 180,E1 12299.006,E2 12299.006} C_VEL
LIN {X 0,Y 268.446,Z 849.651,A -85,B 0,C 180,E1 12295.262,E2 12295.262} C_VEL
LIN {X 0,Y 275.668,Z 836.754,A -85,B 0,C 180,E1 12291.671,E2 12291.671} C_VEL
LIN {X 0,Y 282.822,Z 823.102,A -85,B 0,C 180,E1 12288.62,E2 12288.62} C_VEL
LIN {X 0,Y 290.069,Z 807.949,A -85,B 0,C 180,E1 12285.875,E2 12285.875} C_VEL
LIN {X 0,Y 297.007,Z 791.639,A -85,B 0,C 180,E1 12283.497,E2 12283.497} C_VEL
LIN {X 0,Y 303.333,Z 774.762,A -85,B 0,C 180,E1 12281.495,E2 12281.495} C_VEL
LIN {X 0,Y 309.317,Z 756.217,A -85,B 0,C 180,E1 12279.712,E2 12279.712} C_VEL
LIN {X 0,Y 314.155,Z 738.381,A -85,B 0,C 180,E1 12278.329,E2 12278.329} C_VEL
LIN {X 0,Y 318.419,Z 718.33,A -85,B 0,C 180,E1 12277.107,E2 12277.107} C_VEL
LIN {X 0,Y 321.579,Z 698.236,A -85,B 0,C 180,E1 12276.176,E2 12276.176} C_VEL
LIN {X 0,Y 323.789,Z 676.541,A -85,B 0,C 180,E1 12275.455,E2 12275.455} C_VEL
LIN {X 0,Y 327.968,Z 613.408,A -85,B 0,C 180,E1 12274.113,E2 12274.113} C_VEL
LIN {X 0,Y 327.977,Z 605.836,A -85,B 0,C 180,E1 12273.812,E2 12273.812} C_VEL
LIN {X 0,Y 326.2,Z 586.108,A -85,B 0,C 180,E1 12272.462,E2 12272.462} C_VEL
LIN {X 0,Y 326.297,Z 579.597,A -85,B 0,C 180,E1 12272.217,E2 12272.217} C_VEL
LIN {X 0,Y 330.613,Z 518.778,A -85,B 0,C 180,E1 12270.969,E2 12270.969} C_VEL
LIN {X 0,Y 324.649,Z 508.838,A -85,B 0,C 180,E1 12268.414,E2 12268.414} C_VEL
LIN {X 0,Y 318.351,Z 499.092,A -85,B 0,C 180,E1 12265.336,E2 12265.336} C_VEL
LIN {X 0,Y 313.518,Z 492.167,A -85,B 0,C 180,E1 12262.6,E2 12262.6} C_VEL
LIN {X 0,Y 310.765,Z 488.377,A -85,B 0,C 180,E1 12260.826,E2 12260.826} C_VEL
LIN {X 0,Y 307.581,Z 484.035,A -85,B 0,C 180,E1 12258.479,E2 12258.479} C_VEL
LIN {X 0,Y 304.186,Z 479.517,A -85,B 0,C 180,E1 12255.441,E2 12255.441} C_VEL
LIN {X 0,Y 299.818,Z 474.203,A -85,B 0,C 180,E1 12249.599,E2 12249.599} C_VEL
LIN {X 0,Y 298.192,Z 473.167,A -85,B 0,C 180,E1 12244.616,E2 12244.616} C_VEL
LIN {X 0,Y 298.555,Z 473.916,A -85,B 0,C 180,E1 12239.809,E2 12239.809} C_VEL
LIN {X 0,Y 301.391,Z 479.031,A -85,B 0,C 180,E1 12233.906,E2 12233.906} C_VEL
LIN {X 0,Y 304.728,Z 484.568,A -85,B 0,C 180,E1 12230.081,E2 12230.081} C_VEL
LIN {X 0,Y 307.551,Z 489.07,A -85,B 0,C 180,E1 12227.61,E2 12227.61} C_VEL
LIN {X 0,Y 312.248,Z 496.575,A -85,B 0,C 180,E1 12224.254,E2 12224.254} C_VEL
LIN {X 0,Y 317.269,Z 505.184,A -85,B 0,C 180,E1 12221.25,E2 12221.25} C_VEL
LIN {X 0,Y 323.476,Z 516.253,A -85,B 0,C 180,E1 12218.085,E2 12218.085} C_VEL
LIN {X 0,Y 329.984,Z 528.84,A -85,B 0,C 180,E1 12215.187,E2 12215.187} C_VEL
LIN {X 0,Y 331.658,Z 532.644,A -85,B 0,C 180,E1 12214.475,E2 12214.475} C_VEL
LIN {X 0,Y 316.902,Z 724.393,A -85,B 0,C 180,E1 12210.342,E2 12210.342} C_VEL
LIN {X 0,Y 313.835,Z 746.387,A -85,B 0,C 180,E1 12209.68,E2 12209.68} C_VEL
LIN {X 0,Y 309.205,Z 769.013,A -85,B 0,C 180,E1 12208.784,E2 12208.784} C_VEL
LIN {X 0,Y 303.868,Z 789.354,A -85,B 0,C 180,E1 12207.733,E2 12207.733} C_VEL
LIN {X 0,Y 297.326,Z 810.28,A -85,B 0,C 180,E1 12206.299,E2 12206.299} C_VEL
LIN {X 0,Y 290.2,Z 830.082,A -85,B 0,C 180,E1 12204.543,E2 12204.543} C_VEL
LIN {X 0,Y 282.586,Z 849.122,A -85,B 0,C 180,E1 12202.42,E2 12202.42} C_VEL
LIN {X 0,Y 274.84,Z 866.947,A -85,B 0,C 180,E1 12199.955,E2 12199.955} C_VEL
LIN {X 0,Y 266.945,Z 883.992,A -85,B 0,C 180,E1 12197.025,E2 12197.025} C_VEL
LIN {X 0,Y 259.285,Z 899.876,A -85,B 0,C 180,E1 12193.647,E2 12193.647} C_VEL
LIN {X 0,Y 251.926,Z 915.104,A -85,B 0,C 180,E1 12189.651,E2 12189.651} C_VEL
LIN {X 0,Y 245.668,Z 928.535,A -85,B 0,C 180,E1 12185.302,E2 12185.302} C_VEL
LIN {X 0,Y 240.497,Z 940.623,A -85,B 0,C 180,E1 12180.476,E2 12180.476} C_VEL
LIN {X 0,Y 236.859,Z 950.578,A -85,B 0,C 180,E1 12175.502,E2 12175.502} C_VEL
LIN {X 0,Y 234.633,Z 958.811,A -85,B 0,C 180,E1 12170.366,E2 12170.366} C_VEL
LIN {X 0,Y 233.703,Z 965.109,A -85,B 0,C 180,E1 12165.381,E2 12165.381} C_VEL
LIN {X 0,Y 233.689,Z 969.505,A -85,B 0,C 180,E1 12160.601,E2 12160.601} C_VEL
LIN {X 0,Y 234.127,Z 972.433,A -85,B 0,C 180,E1 12155.883,E2 12155.883} C_VEL
LIN {X 0,Y 234.477,Z 973.575,A -85,B 0,C 180,E1 12151.956,E2 12151.956} C_VEL
LIN {X 0,Y 234.506,Z 973.635,A -85,B 0,C 180,E1 12148.535,E2 12148.535} C_VEL
LIN {X 0,Y 234.224,Z 972.701,A -85,B 0,C 180,E1 12144.858,E2 12144.858} C_VEL
LIN {X 0,Y 233.738,Z 970.079,A -85,B 0,C 180,E1 12140.15,E2 12140.15} C_VEL
LIN {X 0,Y 233.629,Z 966.102,A -85,B 0,C 180,E1 12135.63,E2 12135.63} C_VEL
LIN {X 0,Y 234.445,Z 959.743,A -85,B 0,C 180,E1 12130.314,E2 12130.314} C_VEL
LIN {X 0,Y 236.442,Z 951.933,A -85,B 0,C 180,E1 12125.254,E2 12125.254} C_VEL
LIN {X 0,Y 239.856,Z 942.15,A -85,B 0,C 180,E1 12120.265,E2 12120.265} C_VEL
LIN {X 0,Y 244.502,Z 931.039,A -85,B 0,C 180,E1 12115.649,E2 12115.649} C_VEL
LIN {X 0,Y 250.193,Z 918.719,A -85,B 0,C 180,E1 12111.438,E2 12111.438} C_VEL
LIN {X 0,Y 257.137,Z 904.265,A -85,B 0,C 180,E1 12107.429,E2 12107.429} C_VEL
LIN {X 0,Y 264.566,Z 888.819,A -85,B 0,C 180,E1 12103.957,E2 12103.957} C_VEL
LIN {X 0,Y 272.67,Z 871.465,A -85,B 0,C 180,E1 12100.788,E2 12100.788} C_VEL
LIN {X 0,Y 280.521,Z 853.87,A -85,B 0,C 180,E1 12098.202,E2 12098.202} C_VEL
LIN {X 0,Y 288.21,Z 835.118,A -85,B 0,C 180,E1 12095.985,E2 12095.985} C_VEL
LIN {X 0,Y 295.355,Z 815.696,A -85,B 0,C 180,E1 12094.164,E2 12094.164} C_VEL
LIN {X 0,Y 302.119,Z 794.845,A -85,B 0,C 180,E1 12092.631,E2 12092.631} C_VEL
LIN {X 0,Y 307.754,Z 774.628,A -85,B 0,C 180,E1 12091.49,E2 12091.49} C_VEL
LIN {X 0,Y 312.683,Z 752.41,A -85,B 0,C 180,E1 12090.544,E2 12090.544} C_VEL
LIN {X 0,Y 316.096,Z 730.248,A -85,B 0,C 180,E1 12089.831,E2 12089.831} C_VEL
LIN {X 0,Y 318.82,Z 699.599,A -85,B 0,C 180,E1 12089.108,E2 12089.108} C_VEL
LIN {X 0,Y 331.503,Z 532.098,A -85,B 0,C 180,E1 12085.502,E2 12085.502} C_VEL
LIN {X 0,Y 325.21,Z 519.618,A -85,B 0,C 180,E1 12082.792,E2 12082.792} C_VEL
LIN {X 0,Y 319.028,Z 508.341,A -85,B 0,C 180,E1 12079.784,E2 12079.784} C_VEL
LIN {X 0,Y 313.737,Z 499.326,A -85,B 0,C 180,E1 12076.81,E2 12076.81} C_VEL
LIN {X 0,Y 309.266,Z 491.941,A -85,B 0,C 180,E1 12073.841,E2 12073.841} C_VEL
LIN {X 0,Y 306.056,Z 486.794,A -85,B 0,C 180,E1 12071.304,E2 12071.304} C_VEL
LIN {X 0,Y 303.518,Z 482.8,A -85,B 0,C 180,E1 12068.906,E2 12068.906} C_VEL
LIN {X 0,Y 300.788,Z 478.195,A -85,B 0,C 180,E1 12065.531,E2 12065.531} C_VEL
LIN {X 0,Y 298.269,Z 473.673,A -85,B 0,C 180,E1 12060,E2 12060} C_VEL
LIN {X 0,Y 298.086,Z 473.009,A -85,B 0,C 180,E1 12054.417,E2 12054.417} C_VEL
LIN {X 0,Y 299.967,Z 474.317,A -85,B 0,C 180,E1 12049.63,E2 12049.63} C_VEL
LIN {X 0,Y 304.66,Z 480.184,A -85,B 0,C 180,E1 12043.801,E2 12043.801} C_VEL
LIN {X 0,Y 308.711,Z 485.594,A -85,B 0,C 180,E1 12040.414,E2 12040.414} C_VEL
LIN {X 0,Y 312.583,Z 490.906,A -85,B 0,C 180,E1 12037.774,E2 12037.774} C_VEL
LIN {X 0,Y 317.726,Z 498.191,A -85,B 0,C 180,E1 12034.81,E2 12034.81} C_VEL
LIN {X 0,Y 324.432,Z 508.615,A -85,B 0,C 180,E1 12031.515,E2 12031.515} C_VEL
LIN {X 0,Y 330.449,Z 518.64,A -85,B 0,C 180,E1 12028.942,E2 12028.942} C_VEL
LIN {X 0,Y 327.038,Z 567.309,A -85,B 0,C 180,E1 12027.928,E2 12027.928} C_VEL
LIN {X 0,Y 319.365,Z 677.4,A -85,B 0,C 180,E1 12025.634,E2 12025.634} C_VEL
LIN {X 0,Y 317.087,Z 699.085,A -85,B 0,C 180,E1 12024.913,E2 12024.913} C_VEL
LIN {X 0,Y 313.89,Z 718.906,A -85,B 0,C 180,E1 12023.998,E2 12023.998} C_VEL
LIN {X 0,Y 309.49,Z 739.003,A -85,B 0,C 180,E1 12022.775,E2 12022.775} C_VEL
LIN {X 0,Y 304.214,Z 757.911,A -85,B 0,C 180,E1 12021.306,E2 12021.306} C_VEL
LIN {X 0,Y 298.178,Z 775.957,A -85,B 0,C 180,E1 12019.561,E2 12019.561} C_VEL
LIN {X 0,Y 291.507,Z 793.139,A -85,B 0,C 180,E1 12017.507,E2 12017.507} C_VEL
LIN {X 0,Y 284.35,Z 809.37,A -85,B 0,C 180,E1 12015.116,E2 12015.116} C_VEL
LIN {X 0,Y 277.071,Z 824.049,A -85,B 0,C 180,E1 12012.434,E2 12012.434} C_VEL
LIN {X 0,Y 269.626,Z 837.75,A -85,B 0,C 180,E1 12009.349,E2 12009.349} C_VEL
LIN {X 0,Y 262.084,Z 850.695,A -85,B 0,C 180,E1 12005.706,E2 12005.706} C_VEL
LIN {X 0,Y 255.278,Z 861.733,A -85,B 0,C 180,E1 12001.795,E2 12001.795} C_VEL
LIN {X 0,Y 249.398,Z 871.033,A -85,B 0,C 180,E1 11997.623,E2 11997.623} C_VEL
LIN {X 0,Y 244.158,Z 879.183,A -85,B 0,C 180,E1 11992.867,E2 11992.867} C_VEL
LIN {X 0,Y 240.375,Z 885.175,A -85,B 0,C 180,E1 11988.175,E2 11988.175} C_VEL
LIN {X 0,Y 237.625,Z 889.822,A -85,B 0,C 180,E1 11983.131,E2 11983.131} C_VEL
LIN {X 0,Y 236.01,Z 892.882,A -85,B 0,C 180,E1 11978.035,E2 11978.035} C_VEL
LIN {X 0,Y 235.272,Z 894.473,A -85,B 0,C 180,E1 11972.91,E2 11972.91} C_VEL
LIN {X 0,Y 235.192,Z 894.565,A -85,B 0,C 180,E1 11968.05,E2 11968.05} C_VEL
LIN {X 0,Y 235.796,Z 893.298,A -85,B 0,C 180,E1 11962.862,E2 11962.862} C_VEL
LIN {X 0,Y 237.227,Z 890.64,A -85,B 0,C 180,E1 11957.835,E2 11957.835} C_VEL
LIN {X 0,Y 239.72,Z 886.363,A -85,B 0,C 180,E1 11952.775,E2 11952.775} C_VEL
LIN {X 0,Y 243.471,Z 880.305,A -85,B 0,C 180,E1 11947.803,E2 11947.803} C_VEL
LIN {X 0,Y 248.286,Z 872.775,A -85,B 0,C 180,E1 11943.192,E2 11943.192} C_VEL
LIN {X 0,Y 254.329,Z 863.331,A -85,B 0,C 180,E1 11938.741,E2 11938.741} C_VEL
LIN {X 0,Y 260.806,Z 852.967,A -85,B 0,C 180,E1 11934.899,E2 11934.899} C_VEL
LIN {X 0,Y 267.771,Z 841.258,A -85,B 0,C 180,E1 11931.426,E2 11931.426} C_VEL
LIN {X 0,Y 275.017,Z 828.105,A -85,B 0,C 180,E1 11928.297,E2 11928.297} C_VEL
LIN {X 0,Y 282.404,Z 813.579,A -85,B 0,C 180,E1 11925.496,E2 11925.496} C_VEL
LIN {X 0,Y 289.499,Z 798.137,A -85,B 0,C 180,E1 11923.066,E2 11923.066} C_VEL
LIN {X 0,Y 296.357,Z 781.323,A -85,B 0,C 180,E1 11920.916,E2 11920.916} C_VEL
LIN {X 0,Y 302.627,Z 763.364,A -85,B 0,C 180,E1 11919.072,E2 11919.072} C_VEL
LIN {X 0,Y 307.868,Z 745.567,A -85,B 0,C 180,E1 11917.593,E2 11917.593} C_VEL
LIN {X 0,Y 312.586,Z 725.953,A -85,B 0,C 180,E1 11916.294,E2 11916.294} C_VEL
LIN {X 0,Y 316.272,Z 705.983,A -85,B 0,C 180,E1 11915.268,E2 11915.268} C_VEL
LIN {X 0,Y 318.827,Z 685.517,A -85,B 0,C 180,E1 11914.5,E2 11914.5} C_VEL
LIN {X 0,Y 320.825,Z 657.576,A -85,B 0,C 180,E1 11913.797,E2 11913.797} C_VEL
LIN {X 0,Y 326.297,Z 579.597,A -85,B 0,C 180,E1 11912.217,E2 11912.217} C_VEL
LIN {X 0,Y 326.358,Z 572.027,A -85,B 0,C 180,E1 11911.912,E2 11911.912} C_VEL
LIN {X 0,Y 324.837,Z 552.314,A -85,B 0,C 180,E1 11910.54,E2 11910.54} C_VEL
LIN {X 0,Y 324.983,Z 545.805,A -85,B 0,C 180,E1 11910.293,E2 11910.293} C_VEL
LIN {X 0,Y 326.675,Z 523.209,A -85,B 0,C 180,E1 11909.836,E2 11909.836} C_VEL
LIN {X 0,Y 320.39,Z 512.739,A -85,B 0,C 180,E1 11906.955,E2 11906.955} C_VEL
LIN {X 0,Y 314.626,Z 503.839,A -85,B 0,C 180,E1 11903.903,E2 11903.903} C_VEL
LIN {X 0,Y 309.826,Z 496.712,A -85,B 0,C 180,E1 11900.892,E2 11900.892} C_VEL
LIN {X 0,Y 305.945,Z 491.497,A -85,B 0,C 180,E1 11897.989,E2 11897.989} C_VEL
LIN {X 0,Y 302.86,Z 487.254,A -85,B 0,C 180,E1 11895.119,E2 11895.119} C_VEL
LIN {X 0,Y 298.753,Z 482.097,A -85,B 0,C 180,E1 11889.439,E2 11889.439} C_VEL
LIN {X 0,Y 297.22,Z 481.108,A -85,B 0,C 180,E1 11884.631,E2 11884.631} C_VEL
LIN {X 0,Y 297.574,Z 481.912,A -85,B 0,C 180,E1 11879.808,E2 11879.808} C_VEL
LIN {X 0,Y 300.194,Z 486.862,A -85,B 0,C 180,E1 11874.17,E2 11874.17} C_VEL
LIN {X 0,Y 303.346,Z 492.264,A -85,B 0,C 180,E1 11870.419,E2 11870.419} C_VEL
LIN {X 0,Y 305.973,Z 496.611,A -85,B 0,C 180,E1 11868.024,E2 11868.024} C_VEL
LIN {X 0,Y 310.39,Z 503.942,A -85,B 0,C 180,E1 11864.732,E2 11864.732} C_VEL
LIN {X 0,Y 315.119,Z 512.309,A -85,B 0,C 180,E1 11861.788,E2 11861.788} C_VEL
LIN {X 0,Y 320.99,Z 523.114,A -85,B 0,C 180,E1 11858.675,E2 11858.675} C_VEL
LIN {X 0,Y 327.321,Z 535.766,A -85,B 0,C 180,E1 11855.742,E2 11855.742} C_VEL
LIN {X 0,Y 327.55,Z 536.763,A -85,B 0,C 180,E1 11855.618,E2 11855.618} C_VEL
LIN {X 0,Y 312.657,Z 724.137,A -85,B 0,C 180,E1 11851.583,E2 11851.583} C_VEL
LIN {X 0,Y 309.455,Z 746.113,A -85,B 0,C 180,E1 11850.917,E2 11850.917} C_VEL
LIN {X 0,Y 304.877,Z 767.861,A -85,B 0,C 180,E1 11850.059,E2 11850.059} C_VEL
LIN {X 0,Y 299.222,Z 788.785,A -85,B 0,C 180,E1 11848.984,E2 11848.984} C_VEL
LIN {X 0,Y 292.554,Z 809.466,A -85,B 0,C 180,E1 11847.575,E2 11847.575} C_VEL
LIN {X 0,Y 285.192,Z 829.227,A -85,B 0,C 180,E1 11845.825,E2 11845.825} C_VEL
LIN {X 0,Y 277.275,Z 848.288,A -85,B 0,C 180,E1 11843.695,E2 11843.695} C_VEL
LIN {X 0,Y 269.282,Z 865.981,A -85,B 0,C 180,E1 11841.231,E2 11841.231} C_VEL
LIN {X 0,Y 261.1,Z 882.883,A -85,B 0,C 180,E1 11838.303,E2 11838.303} C_VEL
LIN {X 0,Y 253.243,Z 898.404,A -85,B 0,C 180,E1 11834.965,E2 11834.965} C_VEL
LIN {X 0,Y 245.566,Z 913.492,A -85,B 0,C 180,E1 11830.956,E2 11830.956} C_VEL
LIN {X 0,Y 239.128,Z 926.451,A -85,B 0,C 180,E1 11826.718,E2 11826.718} C_VEL
LIN {X 0,Y 233.499,Z 938.623,A -85,B 0,C 180,E1 11821.78,E2 11821.78} C_VEL
LIN {X 0,Y 229.476,Z 948.692,A -85,B 0,C 180,E1 11816.664,E2 11816.664} C_VEL
LIN {X 0,Y 226.885,Z 957.289,A -85,B 0,C 180,E1 11811.183,E2 11811.183} C_VEL
LIN {X 0,Y 225.797,Z 963.726,A -85,B 0,C 180,E1 11805.934,E2 11805.934} C_VEL
LIN {X 0,Y 225.733,Z 968.141,A -85,B 0,C 180,E1 11800.98,E2 11800.98} C_VEL
LIN {X 0,Y 226.186,Z 971.089,A -85,B 0,C 180,E1 11796.09,E2 11796.09} C_VEL
LIN {X 0,Y 226.579,Z 972.245,A -85,B 0,C 180,E1 11792.024,E2 11792.024} C_VEL
LIN {X 0,Y 226.612,Z 972.305,A -85,B 0,C 180,E1 11788.484,E2 11788.484} C_VEL
LIN {X 0,Y 226.296,Z 971.36,A -85,B 0,C 180,E1 11784.678,E2 11784.678} C_VEL
LIN {X 0,Y 225.782,Z 968.717,A -85,B 0,C 180,E1 11779.799,E2 11779.799} C_VEL
LIN {X 0,Y 225.708,Z 964.721,A -85,B 0,C 180,E1 11775.114,E2 11775.114} C_VEL
LIN {X 0,Y 226.643,Z 958.339,A -85,B 0,C 180,E1 11769.607,E2 11769.607} C_VEL
LIN {X 0,Y 228.856,Z 950.512,A -85,B 0,C 180,E1 11764.376,E2 11764.376} C_VEL
LIN {X 0,Y 232.571,Z 940.717,A -85,B 0,C 180,E1 11759.234,E2 11759.234} C_VEL
LIN {X 0,Y 237.572,Z 929.593,A -85,B 0,C 180,E1 11754.499,E2 11754.499} C_VEL
LIN {X 0,Y 244.007,Z 916.488,A -85,B 0,C 180,E1 11749.965,E2 11749.965} C_VEL
LIN {X 0,Y 251.43,Z 901.956,A -85,B 0,C 180,E1 11745.906,E2 11745.906} C_VEL
LIN {X 0,Y 259.548,Z 885.843,A -85,B 0,C 180,E1 11742.307,E2 11742.307} C_VEL
LIN {X 0,Y 267.557,Z 869.37,A -85,B 0,C 180,E1 11739.334,E2 11739.334} C_VEL
LIN {X 0,Y 276.017,Z 850.992,A -85,B 0,C 180,E1 11736.669,E2 11736.669} C_VEL
LIN {X 0,Y 283.886,Z 832.392,A -85,B 0,C 180,E1 11734.506,E2 11734.506} C_VEL
LIN {X 0,Y 291.374,Z 812.483,A -85,B 0,C 180,E1 11732.686,E2 11732.686} C_VEL
LIN {X 0,Y 297.774,Z 793.098,A -85,B 0,C 180,E1 11731.3,E2 11731.3} C_VEL
LIN {X 0,Y 303.753,Z 771.956,A -85,B 0,C 180,E1 11730.141,E2 11730.141} C_VEL
LIN {X 0,Y 308.67,Z 750.006,A -85,B 0,C 180,E1 11729.229,E2 11729.229} C_VEL
LIN {X 0,Y 312.14,Z 727.411,A -85,B 0,C 180,E1 11728.52,E2 11728.52} C_VEL
LIN {X 0,Y 315.373,Z 689.998,A -85,B 0,C 180,E1 11727.665,E2 11727.665} C_VEL
LIN {X 0,Y 327.42,Z 536.148,A -85,B 0,C 180,E1 11724.368,E2 11724.368} C_VEL
LIN {X 0,Y 321.275,Z 523.822,A -85,B 0,C 180,E1 11721.545,E2 11721.545} C_VEL
LIN {X 0,Y 315.727,Z 513.549,A -85,B 0,C 180,E1 11718.653,E2 11718.653} C_VEL
LIN {X 0,Y 311.487,Z 506.091,A -85,B 0,C 180,E1 11716.12,E2 11716.12} C_VEL
LIN {X 0,Y 307.379,Z 499.109,A -85,B 0,C 180,E1 11713.257,E2 11713.257} C_VEL
LIN {X 0,Y 304.411,Z 494.169,A -85,B 0,C 180,E1 11710.79,E2 11710.79} C_VEL
LIN {X 0,Y 302.071,Z 490.355,A -85,B 0,C 180,E1 11708.47,E2 11708.47} C_VEL
LIN {X 0,Y 299.666,Z 486.066,A -85,B 0,C 180,E1 11705.36,E2 11705.36} C_VEL
LIN {X 0,Y 297.293,Z 481.623,A -85,B 0,C 180,E1 11700,E2 11700} C_VEL
LIN {X 0,Y 297.116,Z 480.951,A -85,B 0,C 180,E1 11694.399,E2 11694.399} C_VEL
LIN {X 0,Y 299.002,Z 482.369,A -85,B 0,C 180,E1 11689.596,E2 11689.596} C_VEL
LIN {X 0,Y 303.318,Z 487.907,A -85,B 0,C 180,E1 11684.121,E2 11684.121} C_VEL
LIN {X 0,Y 307.149,Z 493.165,A -85,B 0,C 180,E1 11680.805,E2 11680.805} C_VEL
LIN {X 0,Y 310.858,Z 498.394,A -85,B 0,C 180,E1 11678.191,E2 11678.191} C_VEL
LIN {X 0,Y 315.806,Z 505.631,A -85,B 0,C 180,E1 11675.246,E2 11675.246} C_VEL
LIN {X 0,Y 322.286,Z 515.945,A -85,B 0,C 180,E1 11671.964,E2 11671.964} C_VEL
LIN {X 0,Y 326.539,Z 523.257,A -85,B 0,C 180,E1 11670.054,E2 11670.054} C_VEL
LIN {X 0,Y 315.23,Z 677.992,A -85,B 0,C 180,E1 11666.866,E2 11666.866} C_VEL
LIN {X 0,Y 312.941,Z 699.354,A -85,B 0,C 180,E1 11666.162,E2 11666.162} C_VEL
LIN {X 0,Y 309.661,Z 719.311,A -85,B 0,C 180,E1 11665.251,E2 11665.251} C_VEL
LIN {X 0,Y 305.116,Z 739.498,A -85,B 0,C 180,E1 11664.03,E2 11664.03} C_VEL
LIN {X 0,Y 300.04,Z 757.34,A -85,B 0,C 180,E1 11662.663,E2 11662.663} C_VEL
LIN {X 0,Y 293.734,Z 775.906,A -85,B 0,C 180,E1 11660.897,E2 11660.897} C_VEL
LIN {X 0,Y 286.969,Z 792.981,A -85,B 0,C 180,E1 11658.886,E2 11658.886} C_VEL
LIN {X 0,Y 279.366,Z 809.709,A -85,B 0,C 180,E1 11656.441,E2 11656.441} C_VEL
LIN {X 0,Y 271.797,Z 824.488,A -85,B 0,C 180,E1 11653.75,E2 11653.75} C_VEL
LIN {X 0,Y 264.023,Z 838.333,A -85,B 0,C 180,E1 11650.639,E2 11650.639} C_VEL
LIN {X 0,Y 256.528,Z 850.753,A -85,B 0,C 180,E1 11647.161,E2 11647.161} C_VEL
LIN {X 0,Y 249.469,Z 861.782,A -85,B 0,C 180,E1 11643.3,E2 11643.3} C_VEL
LIN {X 0,Y 242.796,Z 871.784,A -85,B 0,C 180,E1 11638.8,E2 11638.8} C_VEL
LIN {X 0,Y 237.351,Z 879.758,A -85,B 0,C 180,E1 11634.115,E2 11634.115} C_VEL
LIN {X 0,Y 233.202,Z 885.973,A -85,B 0,C 180,E1 11629.274,E2 11629.274} C_VEL
LIN {X 0,Y 230.026,Z 890.978,A -85,B 0,C 180,E1 11623.829,E2 11623.829} C_VEL
LIN {X 0,Y 228.251,Z 894.115,A -85,B 0,C 180,E1 11618.564,E2 11618.564} C_VEL
LIN {X 0,Y 227.406,Z 895.743,A -85,B 0,C 180,E1 11613.276,E2 11613.276} C_VEL
LIN {X 0,Y 227.296,Z 895.912,A -85,B 0,C 180,E1 11608.235,E2 11608.235} C_VEL
LIN {X 0,Y 227.894,Z 894.756,A -85,B 0,C 180,E1 11602.943,E2 11602.943} C_VEL
LIN {X 0,Y 229.396,Z 892.156,A -85,B 0,C 180,E1 11597.669,E2 11597.669} C_VEL
LIN {X 0,Y 232.152,Z 887.699,A -85,B 0,C 180,E1 11592.195,E2 11592.195} C_VEL
LIN {X 0,Y 236.135,Z 881.645,A -85,B 0,C 180,E1 11587.075,E2 11587.075} C_VEL
LIN {X 0,Y 241.225,Z 874.119,A -85,B 0,C 180,E1 11582.342,E2 11582.342} C_VEL
LIN {X 0,Y 247.58,Z 864.681,A -85,B 0,C 180,E1 11577.789,E2 11577.789} C_VEL
LIN {X 0,Y 254.365,Z 854.327,A -85,B 0,C 180,E1 11573.873,E2 11573.873} C_VEL
LIN {X 0,Y 262.082,Z 841.88,A -85,B 0,C 180,E1 11570.143,E2 11570.143} C_VEL
LIN {X 0,Y 270.093,Z 827.873,A -85,B 0,C 180,E1 11566.826,E2 11566.826} C_VEL
LIN {X 0,Y 277.624,Z 813.404,A -85,B 0,C 180,E1 11564.075,E2 11564.075} C_VEL
LIN {X 0,Y 285.269,Z 797.086,A -85,B 0,C 180,E1 11561.561,E2 11561.561} C_VEL
LIN {X 0,Y 292.426,Z 779.723,A -85,B 0,C 180,E1 11559.406,E2 11559.406} C_VEL
LIN {X 0,Y 298.648,Z 762.288,A -85,B 0,C 180,E1 11557.653,E2 11557.653} C_VEL
LIN {X 0,Y 304.066,Z 743.922,A -85,B 0,C 180,E1 11556.176,E2 11556.176} C_VEL
LIN {X 0,Y 308.774,Z 724.168,A -85,B 0,C 180,E1 11554.916,E2 11554.916} C_VEL
LIN {X 0,Y 312.445,Z 703.794,A -85,B 0,C 180,E1 11553.916,E2 11553.916} C_VEL
LIN {X 0,Y 314.966,Z 683.407,A -85,B 0,C 180,E1 11553.18,E2 11553.18} C_VEL
LIN {X 0,Y 317.862,Z 642.481,A -85,B 0,C 180,E1 11552.243,E2 11552.243} C_VEL
LIN {X 0,Y 324.983,Z 545.805,A -85,B 0,C 180,E1 11550.293,E2 11550.293} C_VEL
LIN {X 0,Y 325.041,Z 539.812,A -85,B 0,C 180,E1 11550.037,E2 11550.037} C_VEL
LIN {X 0,Y 324.292,Z 533.637,A -85,B 0,C 180,E1 11549.483,E2 11549.483} C_VEL
LIN {X 0,Y 322.86,Z 528.372,A -85,B 0,C 180,E1 11548.708,E2 11548.708} C_VEL
LIN {X 0,Y 321.575,Z 525.577,A -85,B 0,C 180,E1 11548.085,E2 11548.085} C_VEL
LIN {X 0,Y 315.693,Z 515.785,A -85,B 0,C 180,E1 11545.113,E2 11545.113} C_VEL
LIN {X 0,Y 310.476,Z 507.713,A -85,B 0,C 180,E1 11542.036,E2 11542.036} C_VEL
LIN {X 0,Y 307.316,Z 503.174,A -85,B 0,C 180,E1 11539.877,E2 11539.877} C_VEL
LIN {X 0,Y 304.553,Z 499.2,A -85,B 0,C 180,E1 11537.679,E2 11537.679} C_VEL
LIN {X 0,Y 301.544,Z 494.989,A -85,B 0,C 180,E1 11534.793,E2 11534.793} C_VEL
LIN {X 0,Y 297.69,Z 489.991,A -85,B 0,C 180,E1 11529.278,E2 11529.278} C_VEL
LIN {X 0,Y 296.225,Z 489.057,A -85,B 0,C 180,E1 11524.453,E2 11524.453} C_VEL
LIN {X 0,Y 296.547,Z 489.785,A -85,B 0,C 180,E1 11520,E2 11520} C_VEL
LIN {X 0,Y 298.997,Z 494.689,A -85,B 0,C 180,E1 11514.435,E2 11514.435} C_VEL
LIN {X 0,Y 301.961,Z 499.955,A -85,B 0,C 180,E1 11510.759,E2 11510.759} C_VEL
LIN {X 0,Y 304.401,Z 504.148,A -85,B 0,C 180,E1 11508.442,E2 11508.442} C_VEL
LIN {X 0,Y 308.492,Z 511.178,A -85,B 0,C 180,E1 11505.261,E2 11505.261} C_VEL
LIN {X 0,Y 313.003,Z 519.433,A -85,B 0,C 180,E1 11502.334,E2 11502.334} C_VEL
LIN {X 0,Y 318.528,Z 529.953,A -85,B 0,C 180,E1 11499.279,E2 11499.279} C_VEL
LIN {X 0,Y 323.605,Z 540.43,A -85,B 0,C 180,E1 11496.797,E2 11496.797} C_VEL
LIN {X 0,Y 308.637,Z 723.119,A -85,B 0,C 180,E1 11492.876,E2 11492.876} C_VEL
LIN {X 0,Y 305.338,Z 745.194,A -85,B 0,C 180,E1 11492.212,E2 11492.212} C_VEL
LIN {X 0,Y 300.516,Z 767.46,A -85,B 0,C 180,E1 11491.337,E2 11491.337} C_VEL
LIN {X 0,Y 294.724,Z 788.22,A -85,B 0,C 180,E1 11490.275,E2 11490.275} C_VEL
LIN {X 0,Y 287.875,Z 808.831,A -85,B 0,C 180,E1 11488.879,E2 11488.879} C_VEL
LIN {X 0,Y 280.292,Z 828.483,A -85,B 0,C 180,E1 11487.141,E2 11487.141} C_VEL
LIN {X 0,Y 272.108,Z 847.453,A -85,B 0,C 180,E1 11485.019,E2 11485.019} C_VEL
LIN {X 0,Y 263.534,Z 865.661,A -85,B 0,C 180,E1 11482.456,E2 11482.456} C_VEL
LIN {X 0,Y 255.048,Z 882.473,A -85,B 0,C 180,E1 11479.506,E2 11479.506} C_VEL
LIN {X 0,Y 246.386,Z 898.762,A -85,B 0,C 180,E1 11475.908,E2 11475.908} C_VEL
LIN {X 0,Y 238.832,Z 912.805,A -85,B 0,C 180,E1 11472.05,E2 11472.05} C_VEL
LIN {X 0,Y 231.723,Z 926.288,A -85,B 0,C 180,E1 11467.471,E2 11467.471} C_VEL
LIN {X 0,Y 226.109,Z 937.757,A -85,B 0,C 180,E1 11462.646,E2 11462.646} C_VEL
LIN {X 0,Y 221.826,Z 947.735,A -85,B 0,C 180,E1 11457.369,E2 11457.369} C_VEL
LIN {X 0,Y 219.145,Z 955.885,A -85,B 0,C 180,E1 11451.969,E2 11451.969} C_VEL
LIN {X 0,Y 217.89,Z 962.411,A -85,B 0,C 180,E1 11446.453,E2 11446.453} C_VEL
LIN {X 0,Y 217.774,Z 966.774,A -85,B 0,C 180,E1 11441.386,E2 11441.386} C_VEL
LIN {X 0,Y 218.212,Z 969.648,A -85,B 0,C 180,E1 11436.578,E2 11436.578} C_VEL
LIN {X 0,Y 218.665,Z 970.882,A -85,B 0,C 180,E1 11432.359,E2 11432.359} C_VEL
LIN {X 0,Y 218.73,Z 971.005,A -85,B 0,C 180,E1 11428.691,E2 11428.691} C_VEL
LIN {X 0,Y 218.399,Z 970.11,A -85,B 0,C 180,E1 11424.748,E2 11424.748} C_VEL
LIN {X 0,Y 217.86,Z 967.745,A -85,B 0,C 180,E1 11419.958,E2 11419.958} C_VEL
LIN {X 0,Y 217.777,Z 963.593,A -85,B 0,C 180,E1 11414.832,E2 11414.832} C_VEL
LIN {X 0,Y 218.703,Z 957.65,A -85,B 0,C 180,E1 11409.392,E2 11409.392} C_VEL
LIN {X 0,Y 221.009,Z 949.93,A -85,B 0,C 180,E1 11403.974,E2 11403.974} C_VEL
LIN {X 0,Y 224.886,Z 940.329,A -85,B 0,C 180,E1 11398.66,E2 11398.66} C_VEL
LIN {X 0,Y 230.722,Z 928.182,A -85,B 0,C 180,E1 11393.293,E2 11393.293} C_VEL
LIN {X 0,Y 237.2,Z 915.797,A -85,B 0,C 180,E1 11388.891,E2 11388.891} C_VEL
LIN {X 0,Y 244.965,Z 901.335,A -85,B 0,C 180,E1 11384.755,E2 11384.755} C_VEL
LIN {X 0,Y 253.167,Z 885.852,A -85,B 0,C 180,E1 11381.213,E2 11381.213} C_VEL
LIN {X 0,Y 261.751,Z 869.042,A -85,B 0,C 180,E1 11378.112,E2 11378.112} C_VEL
LIN {X 0,Y 270.222,Z 851.468,A -85,B 0,C 180,E1 11375.515,E2 11375.515} C_VEL
LIN {X 0,Y 278.327,Z 833.054,A -85,B 0,C 180,E1 11373.341,E2 11373.341} C_VEL
LIN {X 0,Y 285.753,Z 814.194,A -85,B 0,C 180,E1 11371.579,E2 11371.579} C_VEL
LIN {X 0,Y 292.873,Z 793.674,A -85,B 0,C 180,E1 11370.078,E2 11370.078} C_VEL
LIN {X 0,Y 298.992,Z 773.037,A -85,B 0,C 180,E1 11368.929,E2 11368.929} C_VEL
LIN {X 0,Y 304.138,Z 750.972,A -85,B 0,C 180,E1 11368.005,E2 11368.005} C_VEL
LIN {X 0,Y 307.738,Z 729.053,A -85,B 0,C 180,E1 11367.302,E2 11367.302} C_VEL
LIN {X 0,Y 310.607,Z 699.329,A -85,B 0,C 180,E1 11366.598,E2 11366.598} C_VEL
LIN {X 0,Y 323.477,Z 540.286,A -85,B 0,C 180,E1 11363.209,E2 11363.209} C_VEL
LIN {X 0,Y 317.335,Z 527.715,A -85,B 0,C 180,E1 11360.182,E2 11360.182} C_VEL
LIN {X 0,Y 311.411,Z 516.594,A -85,B 0,C 180,E1 11356.796,E2 11356.796} C_VEL
LIN {X 0,Y 306.41,Z 507.688,A -85,B 0,C 180,E1 11353.348,E2 11353.348} C_VEL
LIN {X 0,Y 302.889,Z 501.695,A -85,B 0,C 180,E1 11350.364,E2 11350.364} C_VEL
LIN {X 0,Y 300.642,Z 497.909,A -85,B 0,C 180,E1 11348.029,E2 11348.029} C_VEL
LIN {X 0,Y 298.417,Z 493.796,A -85,B 0,C 180,E1 11344.997,E2 11344.997} C_VEL
LIN {X 0,Y 296.267,Z 489.519,A -85,B 0,C 180,E1 11339.806,E2 11339.806} C_VEL
LIN {X 0,Y 296.145,Z 488.894,A -85,B 0,C 180,E1 11334.381,E2 11334.381} C_VEL
LIN {X 0,Y 297.933,Z 490.27,A -85,B 0,C 180,E1 11329.754,E2 11329.754} C_VEL
LIN {X 0,Y 301.98,Z 495.63,A -85,B 0,C 180,E1 11324.443,E2 11324.443} C_VEL
LIN {X 0,Y 305.714,Z 500.922,A -85,B 0,C 180,E1 11321.108,E2 11321.108} C_VEL
LIN {X 0,Y 309.219,Z 505.987,A -85,B 0,C 180,E1 11318.568,E2 11318.568} C_VEL
LIN {X 0,Y 313.905,Z 513.065,A -85,B 0,C 180,E1 11315.688,E2 11315.688} C_VEL
LIN {X 0,Y 320.425,Z 523.691,A -85,B 0,C 180,E1 11312.293,E2 11312.293} C_VEL
LIN {X 0,Y 322.648,Z 527.89,A -85,B 0,C 180,E1 11311.232,E2 11311.232} C_VEL
LIN {X 0,Y 311.225,Z 678.808,A -85,B 0,C 180,E1 11308.125,E2 11308.125} C_VEL
LIN {X 0,Y 308.891,Z 700.009,A -85,B 0,C 180,E1 11307.428,E2 11307.428} C_VEL
LIN {X 0,Y 305.427,Z 720.437,A -85,B 0,C 180,E1 11306.498,E2 11306.498} C_VEL
LIN {X 0,Y 300.892,Z 739.988,A -85,B 0,C 180,E1 11305.32,E2 11305.32} C_VEL
LIN {X 0,Y 295.585,Z 758.194,A -85,B 0,C 180,E1 11303.936,E2 11303.936} C_VEL
LIN {X 0,Y 289.148,Z 776.635,A -85,B 0,C 180,E1 11302.19,E2 11302.19} C_VEL
LIN {X 0,Y 282.128,Z 793.848,A -85,B 0,C 180,E1 11300.17,E2 11300.17} C_VEL
LIN {X 0,Y 274.272,Z 810.561,A -85,B 0,C 180,E1 11297.727,E2 11297.727} C_VEL
LIN {X 0,Y 266.673,Z 824.927,A -85,B 0,C 180,E1 11295.117,E2 11295.117} C_VEL
LIN {X 0,Y 258.559,Z 838.913,A -85,B 0,C 180,E1 11291.983,E2 11291.983} C_VEL
LIN {X 0,Y 250.703,Z 851.46,A -85,B 0,C 180,E1 11288.469,E2 11288.469} C_VEL
LIN {X 0,Y 243.266,Z 862.585,A -85,B 0,C 180,E1 11284.55,E2 11284.55} C_VEL
LIN {X 0,Y 236.512,Z 872.189,A -85,B 0,C 180,E1 11280.199,E2 11280.199} C_VEL
LIN {X 0,Y 230.636,Z 880.368,A -85,B 0,C 180,E1 11275.412,E2 11275.412} C_VEL
LIN {X 0,Y 225.921,Z 887.041,A -85,B 0,C 180,E1 11270.191,E2 11270.191} C_VEL
LIN {X 0,Y 222.586,Z 891.952,A -85,B 0,C 180,E1 11264.833,E2 11264.833} C_VEL
LIN {X 0,Y 220.576,Z 895.245,A -85,B 0,C 180,E1 11259.39,E2 11259.39} C_VEL
LIN {X 0,Y 219.567,Z 896.953,A -85,B 0,C 180,E1 11253.915,E2 11253.915} C_VEL
LIN {X 0,Y 219.401,Z 897.258,A -85,B 0,C 180,E1 11248.432,E2 11248.432} C_VEL
LIN {X 0,Y 220.004,Z 896.185,A -85,B 0,C 180,E1 11242.951,E2 11242.951} C_VEL
LIN {X 0,Y 221.565,Z 893.659,A -85,B 0,C 180,E1 11237.49,E2 11237.49} C_VEL
LIN {X 0,Y 224.44,Z 889.259,A -85,B 0,C 180,E1 11231.831,E2 11231.831} C_VEL
LIN {X 0,Y 228.376,Z 883.618,A -85,B 0,C 180,E1 11226.796,E2 11226.796} C_VEL
LIN {X 0,Y 233.92,Z 875.881,A -85,B 0,C 180,E1 11221.678,E2 11221.678} C_VEL
LIN {X 0,Y 240.541,Z 866.558,A -85,B 0,C 180,E1 11217.01,E2 11217.01} C_VEL
LIN {X 0,Y 247.592,Z 856.338,A -85,B 0,C 180,E1 11213.011,E2 11213.011} C_VEL
LIN {X 0,Y 255.585,Z 843.983,A -85,B 0,C 180,E1 11209.212,E2 11209.212} C_VEL
LIN {X 0,Y 263.431,Z 830.865,A -85,B 0,C 180,E1 11206.011,E2 11206.011} C_VEL
LIN {X 0,Y 271.65,Z 815.864,A -85,B 0,C 180,E1 11203.067,E2 11203.067} C_VEL
LIN {X 0,Y 279.507,Z 799.86,A -85,B 0,C 180,E1 11200.54,E2 11200.54} C_VEL
LIN {X 0,Y 286.905,Z 782.784,A -85,B 0,C 180,E1 11198.367,E2 11198.367} C_VEL
LIN {X 0,Y 293.605,Z 764.703,A -85,B 0,C 180,E1 11196.523,E2 11196.523} C_VEL
LIN {X 0,Y 299.189,Z 746.667,A -85,B 0,C 180,E1 11195.046,E2 11195.046} C_VEL
LIN {X 0,Y 304.243,Z 726.545,A -85,B 0,C 180,E1 11193.739,E2 11193.739} C_VEL
LIN {X 0,Y 308.064,Z 706.595,A -85,B 0,C 180,E1 11192.738,E2 11192.738} C_VEL
LIN {X 0,Y 310.743,Z 686.267,A -85,B 0,C 180,E1 11191.986,E2 11191.986} C_VEL
LIN {X 0,Y 313.056,Z 655.437,A -85,B 0,C 180,E1 11191.231,E2 11191.231} C_VEL
LIN {X 0,Y 322.783,Z 527.644,A -85,B 0,C 180,E1 11188.644,E2 11188.644} C_VEL
LIN {X 0,Y 321.575,Z 525.577,A -85,B 0,C 180,E1 11188.085,E2 11188.085} C_VEL
LIN {X 0,Y 319.165,Z 522.709,A -85,B 0,C 180,E1 11186.985,E2 11186.985} C_VEL
LIN {X 0,Y 314.726,Z 520.417,A -85,B 0,C 180,E1 11184.946,E2 11184.946} C_VEL
LIN {X 0,Y 310.854,Z 518.165,A -85,B 0,C 180,E1 11182.938,E2 11182.938} C_VEL
LIN {X 0,Y 309.649,Z 516.557,A -85,B 0,C 180,E1 11182.197,E2 11182.197} C_VEL
LIN {X 0,Y 305.868,Z 510.896,A -85,B 0,C 180,E1 11179.577,E2 11179.577} C_VEL
LIN {X 0,Y 303.061,Z 506.78,A -85,B 0,C 180,E1 11177.274,E2 11177.274} C_VEL
LIN {X 0,Y 300.239,Z 502.722,A -85,B 0,C 180,E1 11174.464,E2 11174.464} C_VEL
LIN {X 0,Y 296.63,Z 497.884,A -85,B 0,C 180,E1 11169.116,E2 11169.116} C_VEL
LIN {X 0,Y 295.253,Z 496.997,A -85,B 0,C 180,E1 11164.468,E2 11164.468} C_VEL
LIN {X 0,Y 295.516,Z 497.658,A -85,B 0,C 180,E1 11160.194,E2 11160.194} C_VEL
LIN {X 0,Y 297.802,Z 502.511,A -85,B 0,C 180,E1 11154.703,E2 11154.703} C_VEL
LIN {X 0,Y 300.505,Z 507.478,A -85,B 0,C 180,E1 11151.197,E2 11151.197} C_VEL
LIN {X 0,Y 302.846,Z 511.684,A -85,B 0,C 180,E1 11148.864,E2 11148.864} C_VEL
LIN {X 0,Y 306.744,Z 518.664,A -85,B 0,C 180,E1 11145.706,E2 11145.706} C_VEL
LIN {X 0,Y 310.988,Z 526.695,A -85,B 0,C 180,E1 11142.844,E2 11142.844} C_VEL
LIN {X 0,Y 316.118,Z 536.831,A -85,B 0,C 180,E1 11139.882,E2 11139.882} C_VEL
LIN {X 0,Y 319.752,Z 544.782,A -85,B 0,C 180,E1 11137.993,E2 11137.993} C_VEL
LIN {X 0,Y 304.748,Z 722.396,A -85,B 0,C 180,E1 11134.195,E2 11134.195} C_VEL
LIN {X 0,Y 301.34,Z 744.507,A -85,B 0,C 180,E1 11133.533,E2 11133.533} C_VEL
LIN {X 0,Y 296.541,Z 766.163,A -85,B 0,C 180,E1 11132.691,E2 11132.691} C_VEL
LIN {X 0,Y 290.742,Z 786.56,A -85,B 0,C 180,E1 11131.669,E2 11131.669} C_VEL
LIN {X 0,Y 283.716,Z 807.169,A -85,B 0,C 180,E1 11130.3,E2 11130.3} C_VEL
LIN {X 0,Y 275.894,Z 826.903,A -85,B 0,C 180,E1 11128.583,E2 11128.583} C_VEL
LIN {X 0,Y 267.427,Z 845.925,A -85,B 0,C 180,E1 11126.479,E2 11126.479} C_VEL
LIN {X 0,Y 258.989,Z 863.274,A -85,B 0,C 180,E1 11124.069,E2 11124.069} C_VEL
LIN {X 0,Y 250.067,Z 880.228,A -85,B 0,C 180,E1 11121.117,E2 11121.117} C_VEL
LIN {X 0,Y 241.616,Z 895.473,A -85,B 0,C 180,E1 11117.789,E2 11117.789} C_VEL
LIN {X 0,Y 233.051,Z 910.583,A -85,B 0,C 180,E1 11113.684,E2 11113.684} C_VEL
LIN {X 0,Y 225.562,Z 923.964,A -85,B 0,C 180,E1 11109.13,E2 11109.13} C_VEL
LIN {X 0,Y 219.329,Z 935.75,A -85,B 0,C 180,E1 11104.103,E2 11104.103} C_VEL
LIN {X 0,Y 214.595,Z 945.848,A -85,B 0,C 180,E1 11098.677,E2 11098.677} C_VEL
LIN {X 0,Y 211.414,Z 954.563,A -85,B 0,C 180,E1 11092.747,E2 11092.747} C_VEL
LIN {X 0,Y 209.978,Z 961.21,A -85,B 0,C 180,E1 11086.885,E2 11086.885} C_VEL
LIN {X 0,Y 209.828,Z 965.606,A -85,B 0,C 180,E1 11081.545,E2 11081.545} C_VEL
LIN {X 0,Y 210.34,Z 968.494,A -85,B 0,C 180,E1 11076.277,E2 11076.277} C_VEL
LIN {X 0,Y 210.784,Z 969.584,A -85,B 0,C 180,E1 11072.176,E2 11072.176} C_VEL
LIN {X 0,Y 210.836,Z 969.676,A -85,B 0,C 180,E1 11068.642,E2 11068.642} C_VEL
LIN {X 0,Y 210.501,Z 968.86,A -85,B 0,C 180,E1 11064.824,E2 11064.824} C_VEL
LIN {X 0,Y 209.924,Z 966.547,A -85,B 0,C 180,E1 11059.852,E2 11059.852} C_VEL
LIN {X 0,Y 209.869,Z 962.209,A -85,B 0,C 180,E1 11054.246,E2 11054.246} C_VEL
LIN {X 0,Y 211.034,Z 955.885,A -85,B 0,C 180,E1 11048.315,E2 11048.315} C_VEL
LIN {X 0,Y 213.672,Z 948.098,A -85,B 0,C 180,E1 11042.708,E2 11042.708} C_VEL
LIN {X 0,Y 217.975,Z 938.372,A -85,B 0,C 180,E1 11037.235,E2 11037.235} C_VEL
LIN {X 0,Y 224.01,Z 926.699,A -85,B 0,C 180,E1 11031.984,E2 11031.984} C_VEL
LIN {X 0,Y 231.276,Z 913.667,A -85,B 0,C 180,E1 11027.302,E2 11027.302} C_VEL
LIN {X 0,Y 239.181,Z 899.73,A -85,B 0,C 180,E1 11023.28,E2 11023.28} C_VEL
LIN {X 0,Y 247.983,Z 883.877,A -85,B 0,C 180,E1 11019.645,E2 11019.645} C_VEL
LIN {X 0,Y 256.676,Z 867.541,A -85,B 0,C 180,E1 11016.644,E2 11016.644} C_VEL
LIN {X 0,Y 265.46,Z 849.939,A -85,B 0,C 180,E1 11014.051,E2 11014.051} C_VEL
LIN {X 0,Y 274.152,Z 830.846,A -85,B 0,C 180,E1 11011.824,E2 11011.824} C_VEL
LIN {X 0,Y 281.883,Z 811.636,A -85,B 0,C 180,E1 11010.073,E2 11010.073} C_VEL
LIN {X 0,Y 289.228,Z 790.781,A -85,B 0,C 180,E1 11008.601,E2 11008.601} C_VEL
LIN {X 0,Y 295.568,Z 769.436,A -85,B 0,C 180,E1 11007.469,E2 11007.469} C_VEL
LIN {X 0,Y 300.632,Z 747.715,A -85,B 0,C 180,E1 11006.589,E2 11006.589} C_VEL
LIN {X 0,Y 304.256,Z 725.157,A -85,B 0,C 180,E1 11005.894,E2 11005.894} C_VEL
LIN {X 0,Y 307.758,Z 686.692,A -85,B 0,C 180,E1 11005.025,E2 11005.025} C_VEL
LIN {X 0,Y 319.615,Z 544.328,A -85,B 0,C 180,E1 11002,E2 11002} C_VEL
LIN {X 0,Y 313.784,Z 532.269,A -85,B 0,C 180,E1 10998.918,E2 10998.918} C_VEL
LIN {X 0,Y 308.298,Z 521.692,A -85,B 0,C 180,E1 10995.519,E2 10995.519} C_VEL
LIN {X 0,Y 304.158,Z 514.157,A -85,B 0,C 180,E1 10992.434,E2 10992.434} C_VEL
LIN {X 0,Y 301.289,Z 509.066,A -85,B 0,C 180,E1 10989.84,E2 10989.84} C_VEL
LIN {X 0,Y 299.232,Z 505.462,A -85,B 0,C 180,E1 10987.584,E2 10987.584} C_VEL
LIN {X 0,Y 297.18,Z 501.526,A -85,B 0,C 180,E1 10984.631,E2 10984.631} C_VEL
LIN {X 0,Y 295.237,Z 497.416,A -85,B 0,C 180,E1 10979.611,E2 10979.611} C_VEL
LIN {X 0,Y 295.216,Z 496.853,A -85,B 0,C 180,E1 10974.168,E2 10974.168} C_VEL
LIN {X 0,Y 296.857,Z 498.173,A -85,B 0,C 180,E1 10969.913,E2 10969.913} C_VEL
LIN {X 0,Y 300.739,Z 503.507,A -85,B 0,C 180,E1 10964.674,E2 10964.674} C_VEL
LIN {X 0,Y 304.185,Z 508.491,A -85,B 0,C 180,E1 10961.506,E2 10961.506} C_VEL
LIN {X 0,Y 307.659,Z 513.679,A -85,B 0,C 180,E1 10958.904,E2 10958.904} C_VEL
LIN {X 0,Y 312.098,Z 520.62,A -85,B 0,C 180,E1 10956.092,E2 10956.092} C_VEL
LIN {X 0,Y 318.132,Z 530.759,A -85,B 0,C 180,E1 10952.838,E2 10952.838} C_VEL
LIN {X 0,Y 318.899,Z 532.472,A -85,B 0,C 180,E1 10952.44,E2 10952.44} C_VEL
LIN {X 0,Y 307.388,Z 679.45,A -85,B 0,C 180,E1 10949.42,E2 10949.42} C_VEL
LIN {X 0,Y 305.036,Z 700.403,A -85,B 0,C 180,E1 10948.738,E2 10948.738} C_VEL
LIN {X 0,Y 301.502,Z 720.822,A -85,B 0,C 180,E1 10947.82,E2 10947.82} C_VEL
LIN {X 0,Y 296.826,Z 740.478,A -85,B 0,C 180,E1 10946.646,E2 10946.646} C_VEL
LIN {X 0,Y 291.404,Z 758.671,A -85,B 0,C 180,E1 10945.279,E2 10945.279} C_VEL
LIN {X 0,Y 285.061,Z 776.501,A -85,B 0,C 180,E1 10943.616,E2 10943.616} C_VEL
LIN {X 0,Y 277.633,Z 794.28,A -85,B 0,C 180,E1 10941.555,E2 10941.555} C_VEL
LIN {X 0,Y 269.61,Z 810.83,A -85,B 0,C 180,E1 10939.152,E2 10939.152} C_VEL
LIN {X 0,Y 261.71,Z 825.364,A -85,B 0,C 180,E1 10936.536,E2 10936.536} C_VEL
LIN {X 0,Y 253.246,Z 839.493,A -85,B 0,C 180,E1 10933.385,E2 10933.385} C_VEL
LIN {X 0,Y 245.015,Z 852.165,A -85,B 0,C 180,E1 10929.837,E2 10929.837} C_VEL
LIN {X 0,Y 237.18,Z 863.354,A -85,B 0,C 180,E1 10925.866,E2 10925.866} C_VEL
LIN {X 0,Y 230.027,Z 873.065,A -85,B 0,C 180,E1 10921.435,E2 10921.435} C_VEL
LIN {X 0,Y 223.767,Z 881.345,A -85,B 0,C 180,E1 10916.537,E2 10916.537} C_VEL
LIN {X 0,Y 218.657,Z 888.164,A -85,B 0,C 180,E1 10911.117,E2 10911.117} C_VEL
LIN {X 0,Y 215.072,Z 893.107,A -85,B 0,C 180,E1 10905.64,E2 10905.64} C_VEL
LIN {X 0,Y 212.849,Z 896.442,A -85,B 0,C 180,E1 10900.007,E2 10900.007} C_VEL
LIN {X 0,Y 211.718,Z 898.224,A -85,B 0,C 180,E1 10894.332,E2 10894.332} C_VEL
LIN {X 0,Y 211.507,Z 898.606,A -85,B 0,C 180,E1 10888.645,E2 10888.645} C_VEL
LIN {X 0,Y 212.069,Z 897.712,A -85,B 0,C 180,E1 10883.231,E2 10883.231} C_VEL
LIN {X 0,Y 213.625,Z 895.268,A -85,B 0,C 180,E1 10877.567,E2 10877.567} C_VEL
LIN {X 0,Y 216.395,Z 891.269,A -85,B 0,C 180,E1 10871.967,E2 10871.967} C_VEL
LIN {X 0,Y 220.624,Z 885.592,A -85,B 0,C 180,E1 10866.498,E2 10866.498} C_VEL
LIN {X 0,Y 226.035,Z 878.481,A -85,B 0,C 180,E1 10861.465,E2 10861.465} C_VEL
LIN {X 0,Y 232.807,Z 869.493,A -85,B 0,C 180,E1 10856.654,E2 10856.654} C_VEL
LIN {X 0,Y 240.435,Z 858.908,A -85,B 0,C 180,E1 10852.319,E2 10852.319} C_VEL
LIN {X 0,Y 248.187,Z 847.512,A -85,B 0,C 180,E1 10848.651,E2 10848.651} C_VEL
LIN {X 0,Y 256.745,Z 833.994,A -85,B 0,C 180,E1 10845.185,E2 10845.185} C_VEL
LIN {X 0,Y 265.205,Z 819.379,A -85,B 0,C 180,E1 10842.203,E2 10842.203} C_VEL
LIN {X 0,Y 273.3,Z 803.787,A -85,B 0,C 180,E1 10839.642,E2 10839.642} C_VEL
LIN {X 0,Y 281.027,Z 786.739,A -85,B 0,C 180,E1 10837.405,E2 10837.405} C_VEL
LIN {X 0,Y 288.043,Z 768.848,A -85,B 0,C 180,E1 10835.518,E2 10835.518} C_VEL
LIN {X 0,Y 294.434,Z 749.411,A -85,B 0,C 180,E1 10833.879,E2 10833.879} C_VEL
LIN {X 0,Y 299.608,Z 729.992,A -85,B 0,C 180,E1 10832.587,E2 10832.587} C_VEL
LIN {X 0,Y 303.751,Z 709.733,A -85,B 0,C 180,E1 10831.543,E2 10831.543} C_VEL
LIN {X 0,Y 306.602,Z 689.373,A -85,B 0,C 180,E1 10830.77,E2 10830.77} C_VEL
LIN {X 0,Y 308.81,Z 662.578,A -85,B 0,C 180,E1 10830.075,E2 10830.075} C_VEL
LIN {X 0,Y 319.033,Z 532.232,A -85,B 0,C 180,E1 10827.433,E2 10827.433} C_VEL
LIN {X 0,Y 313.382,Z 522.587,A -85,B 0,C 180,E1 10824.455,E2 10824.455} C_VEL
LIN {X 0,Y 309.649,Z 516.557,A -85,B 0,C 180,E1 10822.197,E2 10822.197} C_VEL
LIN {X 0,Y 307.873,Z 514.598,A -85,B 0,C 180,E1 10821.068,E2 10821.068} C_VEL
LIN {X 0,Y 305.019,Z 513.943,A -85,B 0,C 180,E1 10819.269,E2 10819.269} C_VEL
LIN {X 0,Y 301.425,Z 513.725,A -85,B 0,C 180,E1 10816.68,E2 10816.68} C_VEL
LIN {X 0,Y 300.41,Z 512.771,A -85,B 0,C 180,E1 10815.75,E2 10815.75} C_VEL
LIN {X 0,Y 298.86,Z 510.373,A -85,B 0,C 180,E1 10814.039,E2 10814.039} C_VEL
LIN {X 0,Y 295.571,Z 505.778,A -85,B 0,C 180,E1 10808.953,E2 10808.953} C_VEL
LIN {X 0,Y 294.26,Z 504.947,A -85,B 0,C 180,E1 10804.287,E2 10804.287} C_VEL
LIN {X 0,Y 294.52,Z 505.698,A -85,B 0,C 180,E1 10800.195,E2 10800.195} C_VEL
LIN {X 0,Y 296.62,Z 510.33,A -85,B 0,C 180,E1 10794.972,E2 10794.972} C_VEL
LIN {X 0,Y 299.228,Z 515.334,A -85,B 0,C 180,E1 10791.449,E2 10791.449} C_VEL
LIN {X 0,Y 301.405,Z 519.416,A -85,B 0,C 180,E1 10789.198,E2 10789.198} C_VEL
LIN {X 0,Y 304.962,Z 526.023,A -85,B 0,C 180,E1 10786.201,E2 10786.201} C_VEL
LIN {X 0,Y 308.994,Z 533.954,A -85,B 0,C 180,E1 10783.36,E2 10783.36} C_VEL
LIN {X 0,Y 313.815,Z 543.851,A -85,B 0,C 180,E1 10780.456,E2 10780.456} C_VEL
LIN {X 0,Y 316.06,Z 548.908,A -85,B 0,C 180,E1 10779.221,E2 10779.221} C_VEL
LIN {X 0,Y 301.053,Z 721.428,A -85,B 0,C 180,E1 10775.553,E2 10775.553} C_VEL
LIN {X 0,Y 297.569,Z 743.482,A -85,B 0,C 180,E1 10774.9,E2 10774.9} C_VEL
LIN {X 0,Y 292.663,Z 765.144,A -85,B 0,C 180,E1 10774.069,E2 10774.069} C_VEL
LIN {X 0,Y 286.709,Z 785.585,A -85,B 0,C 180,E1 10773.06,E2 10773.06} C_VEL
LIN {X 0,Y 279.816,Z 805.298,A -85,B 0,C 180,E1 10771.775,E2 10771.775} C_VEL
LIN {X 0,Y 272.041,Z 824.482,A -85,B 0,C 180,E1 10770.149,E2 10770.149} C_VEL
LIN {X 0,Y 262.931,Z 844.398,A -85,B 0,C 180,E1 10767.988,E2 10767.988} C_VEL
LIN {X 0,Y 254.01,Z 862.087,A -85,B 0,C 180,E1 10765.546,E2 10765.546} C_VEL
LIN {X 0,Y 244.468,Z 879.501,A -85,B 0,C 180,E1 10762.503,E2 10762.503} C_VEL
LIN {X 0,Y 235.506,Z 894.919,A -85,B 0,C 180,E1 10759.082,E2 10759.082} C_VEL
LIN {X 0,Y 226.547,Z 909.898,A -85,B 0,C 180,E1 10754.918,E2 10754.918} C_VEL
LIN {X 0,Y 218.923,Z 922.767,A -85,B 0,C 180,E1 10750.428,E2 10750.428} C_VEL
LIN {X 0,Y 212.09,Z 934.89,A -85,B 0,C 180,E1 10745.107,E2 10745.107} C_VEL
LIN {X 0,Y 207.046,Z 944.891,A -85,B 0,C 180,E1 10739.508,E2 10739.508} C_VEL
LIN {X 0,Y 203.654,Z 953.431,A -85,B 0,C 180,E1 10733.432,E2 10733.432} C_VEL
LIN {X 0,Y 202.057,Z 960.096,A -85,B 0,C 180,E1 10727.249,E2 10727.249} C_VEL
LIN {X 0,Y 201.883,Z 964.438,A -85,B 0,C 180,E1 10721.716,E2 10721.716} C_VEL
LIN {X 0,Y 202.399,Z 967.149,A -85,B 0,C 180,E1 10716.524,E2 10716.524} C_VEL
LIN {X 0,Y 202.886,Z 968.254,A -85,B 0,C 180,E1 10712.26,E2 10712.26} C_VEL
LIN {X 0,Y 202.941,Z 968.347,A -85,B 0,C 180,E1 10708.59,E2 10708.59} C_VEL
LIN {X 0,Y 202.561,Z 967.517,A -85,B 0,C 180,E1 10704.62,E2 10704.62} C_VEL
LIN {X 0,Y 201.989,Z 965.336,A -85,B 0,C 180,E1 10699.737,E2 10699.737} C_VEL
LIN {X 0,Y 201.946,Z 961.023,A -85,B 0,C 180,E1 10693.843,E2 10693.843} C_VEL
LIN {X 0,Y 203.214,Z 954.837,A -85,B 0,C 180,E1 10687.741,E2 10687.741} C_VEL
LIN {X 0,Y 206.057,Z 947.092,A -85,B 0,C 180,E1 10681.926,E2 10681.926} C_VEL
LIN {X 0,Y 210.649,Z 937.462,A -85,B 0,C 180,E1 10676.27,E2 10676.27} C_VEL
LIN {X 0,Y 217.037,Z 925.891,A -85,B 0,C 180,E1 10670.872,E2 10670.872} C_VEL
LIN {X 0,Y 224.549,Z 913.219,A -85,B 0,C 180,E1 10666.165,E2 10666.165} C_VEL
LIN {X 0,Y 233.392,Z 898.413,A -85,B 0,C 180,E1 10661.812,E2 10661.812} C_VEL
LIN {X 0,Y 242.43,Z 882.874,A -85,B 0,C 180,E1 10658.217,E2 10658.217} C_VEL
LIN {X 0,Y 251.776,Z 866.039,A -85,B 0,C 180,E1 10655.117,E2 10655.117} C_VEL
LIN {X 0,Y 260.886,Z 848.398,A -85,B 0,C 180,E1 10652.535,E2 10652.535} C_VEL
LIN {X 0,Y 269.88,Z 829.278,A -85,B 0,C 180,E1 10650.331,E2 10650.331} C_VEL
LIN {X 0,Y 277.98,Z 809.69,A -85,B 0,C 180,E1 10648.579,E2 10648.579} C_VEL
LIN {X 0,Y 285.019,Z 790.205,A -85,B 0,C 180,E1 10647.229,E2 10647.229} C_VEL
LIN {X 0,Y 291.439,Z 769.279,A -85,B 0,C 180,E1 10646.127,E2 10646.127} C_VEL
LIN {X 0,Y 296.733,Z 747.246,A -85,B 0,C 180,E1 10645.239,E2 10645.239} C_VEL
LIN {X 0,Y 300.458,Z 724.772,A -85,B 0,C 180,E1 10644.552,E2 10644.552} C_VEL
LIN {X 0,Y 303.771,Z 690.215,A -85,B 0,C 180,E1 10643.768,E2 10643.768} C_VEL
LIN {X 0,Y 315.881,Z 548.552,A -85,B 0,C 180,E1 10640.763,E2 10640.763} C_VEL
LIN {X 0,Y 311.028,Z 538.254,A -85,B 0,C 180,E1 10638.023,E2 10638.023} C_VEL
LIN {X 0,Y 306.197,Z 528.583,A -85,B 0,C 180,E1 10634.852,E2 10634.852} C_VEL
LIN {X 0,Y 302.354,Z 521.322,A -85,B 0,C 180,E1 10631.831,E2 10631.831} C_VEL
LIN {X 0,Y 299.625,Z 516.278,A -85,B 0,C 180,E1 10629.217,E2 10629.217} C_VEL
LIN {X 0,Y 297.764,Z 512.891,A -85,B 0,C 180,E1 10627.04,E2 10627.04} C_VEL
LIN {X 0,Y 295.958,Z 509.255,A -85,B 0,C 180,E1 10624.262,E2 10624.262} C_VEL
LIN {X 0,Y 294.211,Z 505.313,A -85,B 0,C 180,E1 10619.415,E2 10619.415} C_VEL
LIN {X 0,Y 294.245,Z 504.796,A -85,B 0,C 180,E1 10614.149,E2 10614.149} C_VEL
LIN {X 0,Y 295.785,Z 506.078,A -85,B 0,C 180,E1 10610.072,E2 10610.072} C_VEL
LIN {X 0,Y 299.425,Z 511.224,A -85,B 0,C 180,E1 10605.001,E2 10605.001} C_VEL
LIN {X 0,Y 302.665,Z 516.058,A -85,B 0,C 180,E1 10601.908,E2 10601.908} C_VEL
LIN {X 0,Y 305.983,Z 521.163,A -85,B 0,C 180,E1 10599.334,E2 10599.334} C_VEL
LIN {X 0,Y 310.376,Z 528.294,A -85,B 0,C 180,E1 10596.455,E2 10596.455} C_VEL
LIN {X 0,Y 315.306,Z 536.829,A -85,B 0,C 180,E1 10593.681,E2 10593.681} C_VEL
LIN {X 0,Y 303.694,Z 680.312,A -85,B 0,C 180,E1 10590.741,E2 10590.741} C_VEL
LIN {X 0,Y 301.269,Z 701.258,A -85,B 0,C 180,E1 10590.062,E2 10590.062} C_VEL
LIN {X 0,Y 297.576,Z 721.949,A -85,B 0,C 180,E1 10589.136,E2 10589.136} C_VEL
LIN {X 0,Y 292.595,Z 742.216,A -85,B 0,C 180,E1 10587.927,E2 10587.927} C_VEL
LIN {X 0,Y 286.959,Z 760.416,A -85,B 0,C 180,E1 10586.553,E2 10586.553} C_VEL
LIN {X 0,Y 280.115,Z 778.869,A -85,B 0,C 180,E1 10584.816,E2 10584.816} C_VEL
LIN {X 0,Y 272.894,Z 795.564,A -85,B 0,C 180,E1 10582.872,E2 10582.872} C_VEL
LIN {X 0,Y 264.525,Z 812.259,A -85,B 0,C 180,E1 10580.443,E2 10580.443} C_VEL
LIN {X 0,Y 256.345,Z 826.758,A -85,B 0,C 180,E1 10577.816,E2 10577.816} C_VEL
LIN {X 0,Y 247.56,Z 840.867,A -85,B 0,C 180,E1 10574.642,E2 10574.642} C_VEL
LIN {X 0,Y 238.989,Z 853.525,A -85,B 0,C 180,E1 10571.053,E2 10571.053} C_VEL
LIN {X 0,Y 230.803,Z 864.712,A -85,B 0,C 180,E1 10567.019,E2 10567.019} C_VEL
LIN {X 0,Y 223.293,Z 874.415,A -85,B 0,C 180,E1 10562.498,E2 10562.498} C_VEL
LIN {X 0,Y 216.69,Z 882.687,A -85,B 0,C 180,E1 10557.475,E2 10557.475} C_VEL
LIN {X 0,Y 211.316,Z 889.449,A -85,B 0,C 180,E1 10551.947,E2 10551.947} C_VEL
LIN {X 0,Y 207.448,Z 894.443,A -85,B 0,C 180,E1 10546.231,E2 10546.231} C_VEL
LIN {X 0,Y 205.062,Z 897.775,A -85,B 0,C 180,E1 10540.391,E2 10540.391} C_VEL
LIN {X 0,Y 203.847,Z 899.553,A -85,B 0,C 180,E1 10534.5,E2 10534.5} C_VEL
LIN {X 0,Y 203.62,Z 899.934,A -85,B 0,C 180,E1 10528.592,E2 10528.592} C_VEL
LIN {X 0,Y 204.225,Z 899.042,A -85,B 0,C 180,E1 10522.969,E2 10522.969} C_VEL
LIN {X 0,Y 205.897,Z 896.601,A -85,B 0,C 180,E1 10517.093,E2 10517.093} C_VEL
LIN {X 0,Y 208.865,Z 892.605,A -85,B 0,C 180,E1 10511.294,E2 10511.294} C_VEL
LIN {X 0,Y 213.361,Z 886.932,A -85,B 0,C 180,E1 10505.647,E2 10505.647} C_VEL
LIN {X 0,Y 219.093,Z 879.825,A -85,B 0,C 180,E1 10500.473,E2 10500.473} C_VEL
LIN {X 0,Y 226.22,Z 870.841,A -85,B 0,C 180,E1 10495.549,E2 10495.549} C_VEL
LIN {X 0,Y 234.212,Z 860.259,A -85,B 0,C 180,E1 10491.134,E2 10491.134} C_VEL
LIN {X 0,Y 242.301,Z 848.874,A -85,B 0,C 180,E1 10487.414,E2 10487.414} C_VEL
LIN {X 0,Y 251.201,Z 835.373,A -85,B 0,C 180,E1 10483.914,E2 10483.914} C_VEL
LIN {X 0,Y 259.972,Z 820.784,A -85,B 0,C 180,E1 10480.915,E2 10480.915} C_VEL
LIN {X 0,Y 268.342,Z 805.21,A -85,B 0,C 180,E1 10478.347,E2 10478.347} C_VEL
LIN {X 0,Y 276.137,Z 788.612,A -85,B 0,C 180,E1 10476.159,E2 10476.159} C_VEL
LIN {X 0,Y 283.226,Z 771.254,A -85,B 0,C 180,E1 10474.309,E2 10474.309} C_VEL
LIN {X 0,Y 289.478,Z 753.253,A -85,B 0,C 180,E1 10472.756,E2 10472.756} C_VEL
LIN {X 0,Y 295.137,Z 733.232,A -85,B 0,C 180,E1 10471.39,E2 10471.39} C_VEL
LIN {X 0,Y 299.501,Z 712.849,A -85,B 0,C 180,E1 10470.32,E2 10470.32} C_VEL
